LIN {X 0.195,Y -645.562,Z 909.524,A 0.000,B 0.000,C 90.000,E1 130.297} C_DIS
LIN {X -0.083,Y -651.299,Z 909.516,A 0.000,B 0.000,C 90.000,E1 128.830} C_DIS
LIN {X 0.215,Y -657.933,Z 909.506,A 0.000,B 0.000,C 90.000,E1 127.076} C_DIS
LIN {X -0.215,Y -660.619,Z 909.502,A 0.000,B 0.000,C 90.000,E1 126.377} C_DIS
LIN {X -0.067,Y -665.794,Z 909.494,A 0.000,B 0.000,C 90.000,E1 124.898} C_DIS
LIN {X 0.087,Y -669.096,Z 909.488,A 0.000,B 0.000,C 90.000,E1 123.913} C_DIS
LIN {X 0.321,Y -671.422,Z 909.484,A 0.000,B 0.000,C 90.000,E1 123.166} C_DIS
LIN {X 0.173,Y -674.186,Z 909.479,A 0.000,B 0.000,C 90.000,E1 122.212} C_DIS
LIN {X 0.234,Y -677.133,Z 909.472,A 0.000,B 0.000,C 90.000,E1 121.003} C_DIS
LIN {X -0.193,Y -679.151,Z 909.467,A 0.000,B 0.000,C 90.000,E1 120.079} C_DIS
LIN {X 0.332,Y -680.834,Z 909.462,A 0.000,B 0.000,C 90.000,E1 119.077} C_DIS
LIN {X 0.338,Y -682.009,Z 909.458,A 0.000,B 0.000,C 90.000,E1 118.359} C_DIS
LIN {X -0.041,Y -683.207,Z 909.452,A 0.000,B 0.000,C 90.000,E1 117.436} C_DIS
LIN {X -0.114,Y -683.928,Z 909.447,A 0.000,B 0.000,C 90.000,E1 116.488} C_DIS
LIN {X 0.047,Y -684.370,Z 909.441,A 0.000,B 0.000,C 90.000,E1 115.283} C_DIS
LIN {X -0.001,Y -684.293,Z 909.435,A 0.000,B 0.000,C 90.000,E1 114.335} C_DIS
LIN {X 0.425,Y -684.073,Z 909.433,A 0.000,B 0.000,C 90.000,E1 113.823} C_DIS
LIN {X -0.265,Y -683.873,Z 909.431,A 0.000,B 0.000,C 90.000,E1 113.643} C_DIS
LIN {X 0.153,Y -683.084,Z 909.429,A 0.000,B 0.000,C 90.000,E1 113.131} C_DIS
LIN {X 0.093,Y -682.298,Z 909.427,A 0.000,B 0.000,C 90.000,E1 112.898} C_DIS
LIN {X -0.391,Y -680.091,Z 909.425,A 0.000,B 0.000,C 90.000,E1 112.461} C_DIS
LIN {X -0.292,Y -679.235,Z 909.424,A 0.000,B 0.000,C 90.000,E1 112.333} C_DIS
LIN {X -0.194,Y -677.946,Z 909.423,A 0.000,B 0.000,C 90.000,E1 112.206} C_DIS
LIN {X -0.045,Y -676.193,Z 909.423,A 0.000,B 0.000,C 90.000,E1 112.078} C_DIS
LIN {X 0.034,Y -673.633,Z 909.421,A 0.000,B 0.000,C 90.000,E1 111.844} C_DIS
LIN {X 0.216,Y -672.143,Z 909.421,A 0.000,B 0.000,C 90.000,E1 111.716} C_DIS
LIN {X -0.131,Y -669.831,Z 909.420,A 0.000,B 0.000,C 90.000,E1 111.642} C_DIS
LIN {X 0.163,Y -662.934,Z 909.419,A 0.000,B 0.000,C 90.000,E1 111.408} C_DIS
LIN {X 0.168,Y -660.795,Z 909.419,A 0.000,B 0.000,C 90.000,E1 111.354} C_DIS
LIN {X -0.046,Y -652.097,Z 909.418,A 0.000,B 0.000,C 90.000,E1 111.280} C_DIS
LIN {X 0.172,Y -639.351,Z 909.418,A 0.000,B 0.000,C 90.000,E1 111.153} C_DIS
LIN {X -0.202,Y -633.090,Z 909.417,A 0.000,B 0.000,C 90.000,E1 111.099} C_DIS
LIN {X -0.001,Y -627.196,Z 909.417,A 0.000,B 0.000,C 90.000,E1 110.972} C_DIS
LIN {X -0.005,Y -619.742,Z 909.416,A 0.000,B 0.000,C 90.000,E1 110.791} C_DIS
LIN {X 0.025,Y -612.472,Z 909.414,A 0.000,B 0.000,C 90.000,E1 110.556} C_DIS
LIN {X 0.234,Y -605.407,Z 909.413,A 0.000,B 0.000,C 90.000,E1 110.248} C_DIS
LIN {X -0.232,Y -599.446,Z 909.411,A 0.000,B 0.000,C 90.000,E1 109.993} C_DIS
LIN {X 0.123,Y -581.326,Z 909.405,A 0.000,B 0.000,C 90.000,E1 108.852} C_DIS
LIN {X 0.041,Y -577.804,Z 909.404,A 0.000,B 0.000,C 90.000,E1 108.671} C_DIS
LIN {X 0.004,Y -572.696,Z 909.402,A 0.000,B 0.000,C 90.000,E1 108.417} C_DIS
LIN {X -0.230,Y -557.264,Z 909.399,A 0.000,B 0.000,C 90.000,E1 107.819} C_DIS
LIN {X -0.214,Y -556.236,Z 909.399,A 0.000,B 0.000,C 90.000,E1 107.764} C_DIS
LIN {X -0.009,Y -554.802,Z 909.398,A 0.000,B 0.000,C 90.000,E1 107.583} C_DIS
LIN {X -0.049,Y -554.765,Z 909.398,A 0.000,B 0.000,C 90.000,E1 107.583} C_DIS
LIN {X -0.204,Y -554.317,Z 909.396,A 0.000,B 0.000,C 90.000,E1 107.330} C_DIS
LIN {X -0.152,Y -555.407,Z 909.377,A 0.000,B 0.000,C 90.000,E1 103.939} C_DIS
LIN {X 0.224,Y -556.528,Z 909.367,A 0.000,B 0.000,C 90.000,E1 101.951} C_DIS
LIN {X 0.090,Y -557.923,Z 909.356,A 0.000,B 0.000,C 90.000,E1 100.018} C_DIS
LIN {X 0.201,Y -559.105,Z 909.346,A 0.000,B 0.000,C 90.000,E1 98.341} C_DIS
LIN {X 0.275,Y -560.081,Z 909.339,A 0.000,B 0.000,C 90.000,E1 96.947} C_DIS
LIN {X -0.112,Y -561.212,Z 909.328,A 0.000,B 0.000,C 90.000,E1 95.049} C_DIS
LIN {X -0.136,Y -561.882,Z 909.320,A 0.000,B 0.000,C 90.000,E1 93.669} C_DIS
LIN {X -0.082,Y -562.613,Z 909.311,A 0.000,B 0.000,C 90.000,E1 92.007} C_DIS
LIN {X -0.117,Y -563.071,Z 909.303,A 0.000,B 0.000,C 90.000,E1 90.630} C_DIS
LIN {X -0.158,Y -563.456,Z 909.296,A 0.000,B 0.000,C 90.000,E1 89.255} C_DIS
LIN {X -0.073,Y -563.806,Z 909.287,A 0.000,B 0.000,C 90.000,E1 87.593} C_DIS
LIN {X 0.151,Y -564.119,Z 909.276,A 0.000,B 0.000,C 90.000,E1 85.641} C_DIS
LIN {X -0.290,Y -564.432,Z 909.267,A 0.000,B 0.000,C 90.000,E1 84.033} C_DIS
LIN {X 0.199,Y -564.884,Z 909.255,A 0.000,B 0.000,C 90.000,E1 81.781} C_DIS
LIN {X 0.223,Y -565.616,Z 909.242,A 0.000,B 0.000,C 90.000,E1 79.577} C_DIS
LIN {X -0.247,Y -566.559,Z 909.232,A 0.000,B 0.000,C 90.000,E1 77.701} C_DIS
LIN {X -0.007,Y -567.553,Z 909.221,A 0.000,B 0.000,C 90.000,E1 75.755} C_DIS
LIN {X 0.283,Y -568.145,Z 909.215,A 0.000,B 0.000,C 90.000,E1 74.629} C_DIS
LIN {X -0.013,Y -568.893,Z 909.206,A 0.000,B 0.000,C 90.000,E1 73.015} C_DIS
LIN {X 0.078,Y -569.455,Z 909.198,A 0.000,B 0.000,C 90.000,E1 71.638} C_DIS
LIN {X -0.184,Y -569.869,Z 909.190,A 0.000,B 0.000,C 90.000,E1 70.296} C_DIS
LIN {X 0.098,Y -570.165,Z 909.183,A 0.000,B 0.000,C 90.000,E1 68.901} C_DIS
LIN {X 0.230,Y -570.417,Z 909.177,A 0.000,B 0.000,C 90.000,E1 67.794} C_DIS
LIN {X 0.011,Y -570.638,Z 909.168,A 0.000,B 0.000,C 90.000,E1 66.177} C_DIS
LIN {X 0.027,Y -570.717,Z 909.159,A 0.000,B 0.000,C 90.000,E1 64.537} C_DIS
LIN {X -0.048,Y -570.753,Z 909.151,A 0.000,B 0.000,C 90.000,E1 63.179} C_DIS
LIN {X -0.114,Y -570.728,Z 909.143,A 0.000,B 0.000,C 90.000,E1 61.820} C_DIS
LIN {X 0.247,Y -570.545,Z 909.133,A 0.000,B 0.000,C 90.000,E1 59.871} C_DIS
LIN {X 0.070,Y -570.097,Z 909.124,A 0.000,B 0.000,C 90.000,E1 58.250} C_DIS
LIN {X -0.172,Y -569.741,Z 909.119,A 0.000,B 0.000,C 90.000,E1 57.454} C_DIS
LIN {X -0.182,Y -569.052,Z 909.112,A 0.000,B 0.000,C 90.000,E1 56.087} C_DIS
LIN {X 0.114,Y -568.040,Z 909.104,A 0.000,B 0.000,C 90.000,E1 54.689} C_DIS
LIN {X -0.189,Y -567.032,Z 909.098,A 0.000,B 0.000,C 90.000,E1 53.623} C_DIS
LIN {X -0.046,Y -565.386,Z 909.090,A 0.000,B 0.000,C 90.000,E1 52.236} C_DIS
LIN {X -0.057,Y -564.293,Z 909.086,A 0.000,B 0.000,C 90.000,E1 51.412} C_DIS
LIN {X -0.177,Y -563.017,Z 909.081,A 0.000,B 0.000,C 90.000,E1 50.598} C_DIS
LIN {X 0.147,Y -560.951,Z 909.075,A 0.000,B 0.000,C 90.000,E1 49.461} C_DIS
LIN {X -0.095,Y -559.868,Z 909.072,A 0.000,B 0.000,C 90.000,E1 48.933} C_DIS
LIN {X 0.106,Y -557.972,Z 909.067,A 0.000,B 0.000,C 90.000,E1 48.081} C_DIS
LIN {X 0.287,Y -555.739,Z 909.063,A 0.000,B 0.000,C 90.000,E1 47.229} C_DIS
LIN {X 0.006,Y -554.137,Z 909.060,A 0.000,B 0.000,C 90.000,E1 46.701} C_DIS
LIN {X -0.257,Y -551.428,Z 909.055,A 0.000,B 0.000,C 90.000,E1 45.891} C_DIS
LIN {X 0.232,Y -548.426,Z 909.050,A 0.000,B 0.000,C 90.000,E1 45.000} C_DIS
LIN {X -0.086,Y -545.106,Z 909.045,A 0.000,B 0.000,C 90.000,E1 44.190} C_DIS
LIN {X -0.258,Y -543.280,Z 909.043,A 0.000,B 0.000,C 90.000,E1 43.785} C_DIS
LIN {X -0.242,Y -539.229,Z 909.038,A 0.000,B 0.000,C 90.000,E1 42.933} C_DIS
LIN {X 0.313,Y -537.097,Z 909.036,A 0.000,B 0.000,C 90.000,E1 42.447} C_DIS
LIN {X -0.090,Y -534.054,Z 909.033,A 0.000,B 0.000,C 90.000,E1 41.919} C_DIS
LIN {X 0.008,Y -529.937,Z 909.029,A 0.000,B 0.000,C 90.000,E1 41.191} C_DIS
LIN {X -0.040,Y -526.414,Z 909.026,A 0.000,B 0.000,C 90.000,E1 40.620} C_DIS
LIN {X 0.042,Y -521.743,Z 909.022,A 0.000,B 0.000,C 90.000,E1 39.886} C_DIS
LIN {X -0.185,Y -515.782,Z 909.017,A 0.000,B 0.000,C 90.000,E1 39.036} C_DIS
LIN {X -0.320,Y -511.502,Z 909.014,A 0.000,B 0.000,C 90.000,E1 38.463} C_DIS
LIN {X 0.137,Y -508.167,Z 909.011,A 0.000,B 0.000,C 90.000,E1 37.971} C_DIS
LIN {X -0.029,Y -503.410,Z 909.008,A 0.000,B 0.000,C 90.000,E1 37.397} C_DIS
LIN {X -0.153,Y -497.100,Z 909.004,A 0.000,B 0.000,C 90.000,E1 36.664} C_DIS
LIN {X 0.175,Y -490.367,Z 909.000,A 0.000,B 0.000,C 90.000,E1 35.884} C_DIS
LIN {X 0.211,Y -484.732,Z 908.996,A 0.000,B 0.000,C 90.000,E1 35.311} C_DIS
LIN {X 0.108,Y -479.044,Z 908.993,A 0.000,B 0.000,C 90.000,E1 34.771} C_DIS
LIN {X -0.082,Y -473.038,Z 908.990,A 0.000,B 0.000,C 90.000,E1 34.246} C_DIS
LIN {X -0.054,Y -464.073,Z 908.986,A 0.000,B 0.000,C 90.000,E1 33.452} C_DIS
LIN {X -0.014,Y -453.438,Z 908.981,A 0.000,B 0.000,C 90.000,E1 32.546} C_DIS
LIN {X -0.187,Y -442.578,Z 908.976,A 0.000,B 0.000,C 90.000,E1 31.671} C_DIS
LIN {X 0.065,Y -431.669,Z 908.971,A 0.000,B 0.000,C 90.000,E1 30.747} C_DIS
LIN {X -0.085,Y -409.120,Z 908.960,A 0.000,B 0.000,C 90.000,E1 28.743} C_DIS
LIN {X -0.133,Y -398.923,Z 908.954,A 0.000,B 0.000,C 90.000,E1 27.719} C_DIS
LIN {X 0.086,Y -394.402,Z 908.951,A 0.000,B 0.000,C 90.000,E1 27.129} C_DIS
LIN {X -0.030,Y -393.388,Z 908.950,A 0.000,B 0.000,C 90.000,E1 27.001} C_DIS
LIN {X 0.106,Y -390.640,Z 908.947,A 0.000,B 0.000,C 90.000,E1 26.437} C_DIS
LIN {X -0.083,Y -389.421,Z 908.944,A 0.000,B 0.000,C 90.000,E1 25.976} C_DIS
LIN {X -0.231,Y -388.825,Z 908.940,A 0.000,B 0.000,C 90.000,E1 25.283} C_DIS
LIN {X 0.138,Y -388.845,Z 908.936,A 0.000,B 0.000,C 90.000,E1 24.515} C_DIS
LIN {X 0.201,Y -389.687,Z 908.928,A 0.000,B 0.000,C 90.000,E1 23.078} C_DIS
LIN {X -0.187,Y -393.165,Z 908.909,A 0.000,B 0.000,C 90.000,E1 19.577} C_DIS
LIN {X -0.094,Y -396.472,Z 908.893,A 0.000,B 0.000,C 90.000,E1 16.732} C_DIS
LIN {X 0.070,Y -399.567,Z 908.879,A 0.000,B 0.000,C 90.000,E1 14.245} C_DIS
LIN {X -0.159,Y -403.025,Z 908.866,A 0.000,B 0.000,C 90.000,E1 11.827} C_DIS
LIN {X -0.061,Y -407.346,Z 908.850,A 0.000,B 0.000,C 90.000,E1 9.029} C_DIS
LIN {X -0.030,Y -411.518,Z 908.837,A 0.000,B 0.000,C 90.000,E1 6.606} C_DIS
LIN {X 0.125,Y -416.684,Z 908.821,A 0.000,B 0.000,C 90.000,E1 3.841} C_DIS
LIN {X -0.058,Y -422.526,Z 908.806,A 0.000,B 0.000,C 90.000,E1 1.146} C_DIS
LIN {X 0.190,Y -431.613,Z 908.786,A 0.000,B 0.000,C 90.000,E1 357.421} C_DIS
LIN {X -0.066,Y -433.865,Z 908.782,A 0.000,B 0.000,C 90.000,E1 356.788} C_DIS
LIN {X 0.060,Y -436.175,Z 908.779,A 0.000,B 0.000,C 90.000,E1 356.274} C_DIS
LIN {X 0.105,Y -437.112,Z 908.778,A 0.000,B 0.000,C 90.000,E1 356.102} C_DIS
LIN {X 0.134,Y -440.525,Z 908.776,A 0.000,B 0.000,C 90.000,E1 355.698} C_DIS
LIN {X -0.211,Y -442.095,Z 908.775,A 0.000,B 0.000,C 90.000,E1 355.584} C_DIS
LIN {X 0.084,Y -447.635,Z 908.773,A 0.000,B 0.000,C 90.000,E1 355.179} C_DIS
LIN {X -0.204,Y -462.189,Z 908.770,A 0.000,B 0.000,C 90.000,E1 354.546} C_DIS
LIN {X 0.073,Y -475.661,Z 908.766,A 0.000,B 0.000,C 90.000,E1 353.856} C_DIS
LIN {X 0.119,Y -485.730,Z 908.763,A 0.000,B 0.000,C 90.000,E1 353.337} C_DIS
LIN {X 0.093,Y -500.234,Z 908.759,A 0.000,B 0.000,C 90.000,E1 352.534} C_DIS
LIN {X 0.201,Y -508.278,Z 908.756,A 0.000,B 0.000,C 90.000,E1 352.064} C_DIS
LIN {X 0.031,Y -517.662,Z 908.753,A 0.000,B 0.000,C 90.000,E1 351.489} C_DIS
LIN {X 0.171,Y -526.953,Z 908.749,A 0.000,B 0.000,C 90.000,E1 350.849} C_DIS
LIN {X -0.134,Y -532.964,Z 908.747,A 0.000,B 0.000,C 90.000,E1 350.443} C_DIS
LIN {X -0.124,Y -538.715,Z 908.744,A 0.000,B 0.000,C 90.000,E1 349.982} C_DIS
LIN {X 0.185,Y -545.677,Z 908.741,A 0.000,B 0.000,C 90.000,E1 349.342} C_DIS
LIN {X 0.165,Y -552.370,Z 908.737,A 0.000,B 0.000,C 90.000,E1 348.701} C_DIS
LIN {X 0.033,Y -558.750,Z 908.734,A 0.000,B 0.000,C 90.000,E1 348.049} C_DIS
LIN {X -0.138,Y -563.608,Z 908.731,A 0.000,B 0.000,C 90.000,E1 347.521} C_DIS
LIN {X -0.184,Y -570.490,Z 908.726,A 0.000,B 0.000,C 90.000,E1 346.700} C_DIS
LIN {X 0.077,Y -575.709,Z 908.722,A 0.000,B 0.000,C 90.000,E1 345.992} C_DIS
LIN {X -0.070,Y -579.705,Z 908.719,A 0.000,B 0.000,C 90.000,E1 345.463} C_DIS
LIN {X -0.144,Y -586.930,Z 908.713,A 0.000,B 0.000,C 90.000,E1 344.393} C_DIS
LIN {X -0.301,Y -591.105,Z 908.710,A 0.000,B 0.000,C 90.000,E1 343.740} C_DIS
LIN {X -0.047,Y -597.242,Z 908.704,A 0.000,B 0.000,C 90.000,E1 342.653} C_DIS
LIN {X 0.113,Y -602.926,Z 908.698,A 0.000,B 0.000,C 90.000,E1 341.583} C_DIS
LIN {X -0.074,Y -608.917,Z 908.691,A 0.000,B 0.000,C 90.000,E1 340.423} C_DIS
LIN {X -0.120,Y -613.345,Z 908.686,A 0.000,B 0.000,C 90.000,E1 339.518} C_DIS
LIN {X 0.097,Y -617.537,Z 908.681,A 0.000,B 0.000,C 90.000,E1 338.592} C_DIS
LIN {X 0.110,Y -623.248,Z 908.674,A 0.000,B 0.000,C 90.000,E1 337.305} C_DIS
LIN {X -0.133,Y -627.339,Z 908.668,A 0.000,B 0.000,C 90.000,E1 336.305} C_DIS
LIN {X -0.060,Y -631.107,Z 908.663,A 0.000,B 0.000,C 90.000,E1 335.281} C_DIS
LIN {X -0.198,Y -634.766,Z 908.657,A 0.000,B 0.000,C 90.000,E1 334.280} C_DIS
LIN {X -0.066,Y -637.407,Z 908.653,A 0.000,B 0.000,C 90.000,E1 333.512} C_DIS
LIN {X 0.094,Y -639.777,Z 908.649,A 0.000,B 0.000,C 90.000,E1 332.743} C_DIS
LIN {X -0.225,Y -642.799,Z 908.643,A 0.000,B 0.000,C 90.000,E1 331.769} C_DIS
LIN {X 0.371,Y -645.562,Z 908.638,A 0.000,B 0.000,C 90.000,E1 330.717} C_DIS
LIN {X -0.357,Y -648.851,Z 908.631,A 0.000,B 0.000,C 90.000,E1 329.537} C_DIS
LIN {X -0.155,Y -651.906,Z 908.624,A 0.000,B 0.000,C 90.000,E1 328.280} C_DIS
LIN {X -0.096,Y -653.633,Z 908.620,A 0.000,B 0.000,C 90.000,E1 327.533} C_DIS
LIN {X -0.023,Y -655.966,Z 908.613,A 0.000,B 0.000,C 90.000,E1 326.294} C_DIS
LIN {X 0.074,Y -657.235,Z 908.609,A 0.000,B 0.000,C 90.000,E1 325.548} C_DIS
LIN {X 0.043,Y -658.966,Z 908.602,A 0.000,B 0.000,C 90.000,E1 324.322} C_DIS
LIN {X -0.338,Y -660.459,Z 908.595,A 0.000,B 0.000,C 90.000,E1 323.130} C_DIS
LIN {X 0.178,Y -661.956,Z 908.587,A 0.000,B 0.000,C 90.000,E1 321.618} C_DIS
LIN {X 0.177,Y -663.531,Z 908.577,A 0.000,B 0.000,C 90.000,E1 319.908} C_DIS
LIN {X 0.182,Y -665.606,Z 908.565,A 0.000,B 0.000,C 90.000,E1 317.715} C_DIS
LIN {X -0.293,Y -666.828,Z 908.558,A 0.000,B 0.000,C 90.000,E1 316.539} C_DIS
LIN {X -0.290,Y -667.514,Z 908.554,A 0.000,B 0.000,C 90.000,E1 315.810} C_DIS
LIN {X -0.253,Y -669.043,Z 908.545,A 0.000,B 0.000,C 90.000,E1 314.109} C_DIS
LIN {X 0.296,Y -670.591,Z 908.536,A 0.000,B 0.000,C 90.000,E1 312.366} C_DIS
LIN {X 0.400,Y -671.731,Z 908.529,A 0.000,B 0.000,C 90.000,E1 311.148} C_DIS
LIN {X 0.098,Y -672.889,Z 908.521,A 0.000,B 0.000,C 90.000,E1 309.725} C_DIS
LIN {X -0.191,Y -673.865,Z 908.514,A 0.000,B 0.000,C 90.000,E1 308.543} C_DIS
LIN {X 0.064,Y -674.800,Z 908.507,A 0.000,B 0.000,C 90.000,E1 307.317} C_DIS
LIN {X -0.207,Y -675.377,Z 908.502,A 0.000,B 0.000,C 90.000,E1 306.377} C_DIS
LIN {X 0.214,Y -676.122,Z 908.494,A 0.000,B 0.000,C 90.000,E1 304.898} C_DIS
LIN {X -0.296,Y -676.820,Z 908.486,A 0.000,B 0.000,C 90.000,E1 303.499} C_DIS
LIN {X -0.064,Y -677.837,Z 908.477,A 0.000,B 0.000,C 90.000,E1 301.799} C_DIS
LIN {X 0.028,Y -679.350,Z 908.466,A 0.000,B 0.000,C 90.000,E1 299.873} C_DIS
LIN {X 0.257,Y -682.866,Z 908.449,A 0.000,B 0.000,C 90.000,E1 296.744} C_DIS
LIN {X 0.145,Y -685.537,Z 908.438,A 0.000,B 0.000,C 90.000,E1 294.847} C_DIS
LIN {X 0.116,Y -686.627,Z 908.433,A 0.000,B 0.000,C 90.000,E1 293.898} C_DIS
LIN {X -0.075,Y -687.047,Z 908.430,A 0.000,B 0.000,C 90.000,E1 293.439} C_DIS
LIN {X 0.093,Y -687.264,Z 908.428,A 0.000,B 0.000,C 90.000,E1 292.950} C_DIS
LIN {X 0.265,Y -686.844,Z 908.425,A 0.000,B 0.000,C 90.000,E1 292.461} C_DIS
LIN {X -0.153,Y -686.411,Z 908.424,A 0.000,B 0.000,C 90.000,E1 292.259} C_DIS
LIN {X 0.015,Y -684.112,Z 908.421,A 0.000,B 0.000,C 90.000,E1 291.770} C_DIS
LIN {X -0.029,Y -682.572,Z 908.420,A 0.000,B 0.000,C 90.000,E1 291.535} C_DIS
LIN {X 0.071,Y -681.425,Z 908.419,A 0.000,B 0.000,C 90.000,E1 291.408} C_DIS
LIN {X 0.170,Y -679.661,Z 908.418,A 0.000,B 0.000,C 90.000,E1 291.280} C_DIS
LIN {X 0.158,Y -672.887,Z 908.416,A 0.000,B 0.000,C 90.000,E1 290.918} C_DIS
LIN {X 0.153,Y -665.738,Z 908.415,A 0.000,B 0.000,C 90.000,E1 290.610} C_DIS
LIN {X 0.151,Y -661.194,Z 908.413,A 0.000,B 0.000,C 90.000,E1 290.375} C_DIS
LIN {X 0.091,Y -661.149,Z 908.413,A 0.000,B 0.000,C 90.000,E1 290.375} C_DIS
LIN {X -0.048,Y -660.567,Z 908.413,A 0.000,B 0.000,C 90.000,E1 290.301} C_DIS
LIN {X -0.093,Y -660.547,Z 908.413,A 0.000,B 0.000,C 90.000,E1 290.301} C_DIS
LIN {X 0.061,Y -660.564,Z 908.412,A 0.000,B 0.000,C 90.000,E1 290.066} C_DIS
LIN {X 0.064,Y -662.013,Z 908.409,A 0.000,B 0.000,C 90.000,E1 289.577} C_DIS
LIN {X 0.151,Y -664.034,Z 908.406,A 0.000,B 0.000,C 90.000,E1 289.087} C_DIS
LIN {X 0.047,Y -671.509,Z 908.398,A 0.000,B 0.000,C 90.000,E1 287.638} C_DIS
LIN {X -0.090,Y -673.798,Z 908.395,A 0.000,B 0.000,C 90.000,E1 287.166} C_DIS
LIN {X -0.072,Y -676.837,Z 908.391,A 0.000,B 0.000,C 90.000,E1 286.441} C_DIS
LIN {X -0.031,Y -679.173,Z 908.387,A 0.000,B 0.000,C 90.000,E1 285.717} C_DIS
LIN {X -0.117,Y -680.451,Z 908.385,A 0.000,B 0.000,C 90.000,E1 285.245} C_DIS
LIN {X -0.287,Y -683.062,Z 908.378,A 0.000,B 0.000,C 90.000,E1 284.064} C_DIS
LIN {X 0.297,Y -684.275,Z 908.374,A 0.000,B 0.000,C 90.000,E1 283.300} C_DIS
LIN {X 0.205,Y -685.582,Z 908.369,A 0.000,B 0.000,C 90.000,E1 282.355} C_DIS
LIN {X 0.000,Y -686.195,Z 908.365,A 0.000,B 0.000,C 90.000,E1 281.658} C_DIS
LIN {X -0.039,Y -686.413,Z 908.362,A 0.000,B 0.000,C 90.000,E1 281.186} C_DIS
LIN {X -0.082,Y -686.381,Z 908.360,A 0.000,B 0.000,C 90.000,E1 280.715} C_DIS
LIN {X -0.251,Y -685.980,Z 908.357,A 0.000,B 0.000,C 90.000,E1 280.254} C_DIS
LIN {X -0.275,Y -685.653,Z 908.356,A 0.000,B 0.000,C 90.000,E1 280.018} C_DIS
LIN {X 0.232,Y -684.729,Z 908.353,A 0.000,B 0.000,C 90.000,E1 279.500} C_DIS
LIN {X 0.170,Y -683.507,Z 908.350,A 0.000,B 0.000,C 90.000,E1 279.029} C_DIS
LIN {X -0.008,Y -681.823,Z 908.348,A 0.000,B 0.000,C 90.000,E1 278.568} C_DIS
LIN {X -0.194,Y -679.778,Z 908.345,A 0.000,B 0.000,C 90.000,E1 278.106} C_DIS
LIN {X 0.223,Y -676.392,Z 908.341,A 0.000,B 0.000,C 90.000,E1 277.352} C_DIS
LIN {X -0.075,Y -673.192,Z 908.338,A 0.000,B 0.000,C 90.000,E1 276.777} C_DIS
LIN {X 0.271,Y -669.663,Z 908.334,A 0.000,B 0.000,C 90.000,E1 276.144} C_DIS
LIN {X 0.093,Y -667.413,Z 908.332,A 0.000,B 0.000,C 90.000,E1 275.796} C_DIS
LIN {X -0.272,Y -663.096,Z 908.329,A 0.000,B 0.000,C 90.000,E1 275.220} C_DIS
LIN {X 0.081,Y -659.326,Z 908.326,A 0.000,B 0.000,C 90.000,E1 274.702} C_DIS
LIN {X -0.299,Y -655.183,Z 908.323,A 0.000,B 0.000,C 90.000,E1 274.245} C_DIS
LIN {X -0.107,Y -649.293,Z 908.320,A 0.000,B 0.000,C 90.000,E1 273.612} C_DIS
LIN {X 0.291,Y -644.297,Z 908.317,A 0.000,B 0.000,C 90.000,E1 273.094} C_DIS
LIN {X 0.278,Y -637.563,Z 908.314,A 0.000,B 0.000,C 90.000,E1 272.522} C_DIS
LIN {X -0.070,Y -630.336,Z 908.311,A 0.000,B 0.000,C 90.000,E1 272.007} C_DIS
LIN {X -0.095,Y -624.332,Z 908.309,A 0.000,B 0.000,C 90.000,E1 271.604} C_DIS
LIN {X 0.089,Y -618.139,Z 908.307,A 0.000,B 0.000,C 90.000,E1 271.203} C_DIS
LIN {X 0.255,Y -609.882,Z 908.304,A 0.000,B 0.000,C 90.000,E1 270.745} C_DIS
LIN {X -0.185,Y -603.169,Z 908.302,A 0.000,B 0.000,C 90.000,E1 270.458} C_DIS
LIN {X -0.219,Y -598.145,Z 908.301,A 0.000,B 0.000,C 90.000,E1 270.229} C_DIS
LIN {X -0.149,Y -590.978,Z 908.300,A 0.000,B 0.000,C 90.000,E1 269.943} C_DIS
LIN {X 0.259,Y -583.781,Z 908.298,A 0.000,B 0.000,C 90.000,E1 269.656} C_DIS
LIN {X -0.249,Y -578.196,Z 908.297,A 0.000,B 0.000,C 90.000,E1 269.542} C_DIS
LIN {X 0.036,Y -571.792,Z 908.297,A 0.000,B 0.000,C 90.000,E1 269.370} C_DIS
LIN {X 0.144,Y -565.261,Z 908.296,A 0.000,B 0.000,C 90.000,E1 269.255} C_DIS
LIN {X -0.224,Y -554.852,Z 908.295,A 0.000,B 0.000,C 90.000,E1 269.198} C_DIS
LIN {X 0.157,Y -552.543,Z 908.295,A 0.000,B 0.000,C 90.000,E1 269.141} C_DIS
LIN {X -0.136,Y -549.494,Z 908.295,A 0.000,B 0.000,C 90.000,E1 269.083} C_DIS
LIN {X -0.168,Y -549.414,Z 908.295,A 0.000,B 0.000,C 90.000,E1 269.083} C_DIS
LIN {X 0.187,Y -545.395,Z 908.293,A 0.000,B 0.000,C 90.000,E1 268.682} C_DIS
LIN {X 0.150,Y -545.361,Z 908.293,A 0.000,B 0.000,C 90.000,E1 268.682} C_DIS
LIN {X 0.055,Y -544.265,Z 908.291,A 0.000,B 0.000,C 90.000,E1 268.396} C_DIS
LIN {X -0.029,Y -543.383,Z 908.288,A 0.000,B 0.000,C 90.000,E1 267.822} C_DIS
LIN {X -0.155,Y -540.427,Z 908.269,A 0.000,B 0.000,C 90.000,E1 264.432} C_DIS
LIN {X -0.017,Y -539.422,Z 908.261,A 0.000,B 0.000,C 90.000,E1 262.996} C_DIS
LIN {X 0.167,Y -538.477,Z 908.255,A 0.000,B 0.000,C 90.000,E1 261.837} C_DIS
LIN {X -0.128,Y -537.130,Z 908.247,A 0.000,B 0.000,C 90.000,E1 260.443} C_DIS
LIN {X 0.020,Y -535.946,Z 908.241,A 0.000,B 0.000,C 90.000,E1 259.285} C_DIS
LIN {X 0.190,Y -535.031,Z 908.236,A 0.000,B 0.000,C 90.000,E1 258.409} C_DIS
LIN {X 0.046,Y -533.384,Z 908.228,A 0.000,B 0.000,C 90.000,E1 256.992} C_DIS
LIN {X -0.077,Y -531.258,Z 908.218,A 0.000,B 0.000,C 90.000,E1 255.283} C_DIS
LIN {X 0.079,Y -528.397,Z 908.205,A 0.000,B 0.000,C 90.000,E1 252.960} C_DIS
LIN {X 0.120,Y -526.617,Z 908.197,A 0.000,B 0.000,C 90.000,E1 251.511} C_DIS
LIN {X 0.294,Y -524.330,Z 908.188,A 0.000,B 0.000,C 90.000,E1 249.752} C_DIS
LIN {X 0.273,Y -522.809,Z 908.181,A 0.000,B 0.000,C 90.000,E1 248.592} C_DIS
LIN {X -0.107,Y -520.766,Z 908.173,A 0.000,B 0.000,C 90.000,E1 247.177} C_DIS
LIN {X 0.006,Y -519.133,Z 908.167,A 0.000,B 0.000,C 90.000,E1 245.997} C_DIS
LIN {X 0.117,Y -515.655,Z 908.154,A 0.000,B 0.000,C 90.000,E1 243.640} C_DIS
LIN {X -0.093,Y -512.723,Z 908.144,A 0.000,B 0.000,C 90.000,E1 241.897} C_DIS
LIN {X -0.104,Y -510.600,Z 908.137,A 0.000,B 0.000,C 90.000,E1 240.717} C_DIS
LIN {X 0.138,Y -506.936,Z 908.126,A 0.000,B 0.000,C 90.000,E1 238.614} C_DIS
LIN {X -0.138,Y -504.719,Z 908.119,A 0.000,B 0.000,C 90.000,E1 237.454} C_DIS
LIN {X 0.254,Y -502.306,Z 908.112,A 0.000,B 0.000,C 90.000,E1 236.215} C_DIS
LIN {X 0.032,Y -500.378,Z 908.108,A 0.000,B 0.000,C 90.000,E1 235.341} C_DIS
LIN {X 0.230,Y -497.545,Z 908.101,A 0.000,B 0.000,C 90.000,E1 234.116} C_DIS
LIN {X 0.099,Y -494.880,Z 908.094,A 0.000,B 0.000,C 90.000,E1 232.924} C_DIS
LIN {X 0.069,Y -491.502,Z 908.086,A 0.000,B 0.000,C 90.000,E1 231.412} C_DIS
LIN {X -0.114,Y -486.769,Z 908.074,A 0.000,B 0.000,C 90.000,E1 229.299} C_DIS
LIN {X 0.002,Y -484.753,Z 908.069,A 0.000,B 0.000,C 90.000,E1 228.366} C_DIS
LIN {X 0.091,Y -479.245,Z 908.055,A 0.000,B 0.000,C 90.000,E1 225.891} C_DIS
LIN {X 0.003,Y -475.753,Z 908.046,A 0.000,B 0.000,C 90.000,E1 224.352} C_DIS
LIN {X 0.188,Y -472.164,Z 908.038,A 0.000,B 0.000,C 90.000,E1 222.771} C_DIS
LIN {X -0.176,Y -467.264,Z 908.026,A 0.000,B 0.000,C 90.000,E1 220.620} C_DIS
LIN {X -0.122,Y -463.916,Z 908.017,A 0.000,B 0.000,C 90.000,E1 219.036} C_DIS
LIN {X 0.046,Y -459.878,Z 908.006,A 0.000,B 0.000,C 90.000,E1 217.111} C_DIS
LIN {X 0.025,Y -456.526,Z 907.997,A 0.000,B 0.000,C 90.000,E1 215.518} C_DIS
LIN {X 0.037,Y -453.105,Z 907.988,A 0.000,B 0.000,C 90.000,E1 213.913} C_DIS
LIN {X -0.030,Y -447.336,Z 907.974,A 0.000,B 0.000,C 90.000,E1 211.337} C_DIS
LIN {X 0.185,Y -445.182,Z 907.969,A 0.000,B 0.000,C 90.000,E1 210.335} C_DIS
LIN {X -0.076,Y -440.957,Z 907.958,A 0.000,B 0.000,C 90.000,E1 208.409} C_DIS
LIN {X 0.095,Y -437.328,Z 907.949,A 0.000,B 0.000,C 90.000,E1 206.744} C_DIS
LIN {X 0.018,Y -432.988,Z 907.938,A 0.000,B 0.000,C 90.000,E1 204.771} C_DIS
LIN {X 0.051,Y -428.640,Z 907.927,A 0.000,B 0.000,C 90.000,E1 202.770} C_DIS
LIN {X 0.021,Y -425.079,Z 907.917,A 0.000,B 0.000,C 90.000,E1 201.099} C_DIS
LIN {X -0.054,Y -420.844,Z 907.906,A 0.000,B 0.000,C 90.000,E1 199.087} C_DIS
LIN {X -0.127,Y -417.501,Z 907.897,A 0.000,B 0.000,C 90.000,E1 197.402} C_DIS
LIN {X -0.238,Y -413.381,Z 907.885,A 0.000,B 0.000,C 90.000,E1 195.371} C_DIS
LIN {X -0.044,Y -408.578,Z 907.872,A 0.000,B 0.000,C 90.000,E1 192.939} C_DIS
LIN {X 0.107,Y -405.900,Z 907.864,A 0.000,B 0.000,C 90.000,E1 191.535} C_DIS
LIN {X 0.144,Y -402.449,Z 907.855,A 0.000,B 0.000,C 90.000,E1 189.792} C_DIS
LIN {X 0.098,Y -398.212,Z 907.843,A 0.000,B 0.000,C 90.000,E1 187.701} C_DIS
LIN {X 0.070,Y -392.221,Z 907.825,A 0.000,B 0.000,C 90.000,E1 184.531} C_DIS
LIN {X -0.089,Y -388.034,Z 907.811,A 0.000,B 0.000,C 90.000,E1 182.064} C_DIS
LIN {X -0.170,Y -385.133,Z 907.802,A 0.000,B 0.000,C 90.000,E1 180.286} C_DIS
LIN {X -0.153,Y -381.252,Z 907.787,A 0.000,B 0.000,C 90.000,E1 177.764} C_DIS
LIN {X 0.031,Y -378.681,Z 907.777,A 0.000,B 0.000,C 90.000,E1 175.927} C_DIS
LIN {X 0.032,Y -377.484,Z 907.771,A 0.000,B 0.000,C 90.000,E1 174.837} C_DIS
LIN {X -0.056,Y -376.839,Z 907.763,A 0.000,B 0.000,C 90.000,E1 173.394} C_DIS
LIN {X 0.166,Y -376.923,Z 907.761,A 0.000,B 0.000,C 90.000,E1 172.996} C_DIS
LIN {X 0.060,Y -377.171,Z 907.759,A 0.000,B 0.000,C 90.000,E1 172.648} C_DIS
LIN {X -0.151,Y -378.296,Z 907.755,A 0.000,B 0.000,C 90.000,E1 171.951} C_DIS
LIN {X 0.123,Y -379.387,Z 907.753,A 0.000,B 0.000,C 90.000,E1 171.546} C_DIS
LIN {X -0.069,Y -381.425,Z 907.749,A 0.000,B 0.000,C 90.000,E1 170.849} C_DIS
LIN {X -0.180,Y -384.461,Z 907.746,A 0.000,B 0.000,C 90.000,E1 170.330} C_DIS
LIN {X 0.105,Y -387.519,Z 907.744,A 0.000,B 0.000,C 90.000,E1 169.859} C_DIS
LIN {X -0.121,Y -393.894,Z 907.740,A 0.000,B 0.000,C 90.000,E1 169.275} C_DIS
LIN {X 0.004,Y -401.829,Z 907.737,A 0.000,B 0.000,C 90.000,E1 168.701} C_DIS
LIN {X 0.222,Y -407.065,Z 907.735,A 0.000,B 0.000,C 90.000,E1 168.342} C_DIS
LIN {X -0.223,Y -418.459,Z 907.731,A 0.000,B 0.000,C 90.000,E1 167.645} C_DIS
LIN {X -0.041,Y -424.881,Z 907.729,A 0.000,B 0.000,C 90.000,E1 167.173} C_DIS
LIN {X 0.009,Y -431.295,Z 907.726,A 0.000,B 0.000,C 90.000,E1 166.700} C_DIS
LIN {X -0.224,Y -439.099,Z 907.723,A 0.000,B 0.000,C 90.000,E1 166.117} C_DIS
LIN {X -0.202,Y -452.668,Z 907.716,A 0.000,B 0.000,C 90.000,E1 164.936} C_DIS
LIN {X -0.153,Y -461.243,Z 907.712,A 0.000,B 0.000,C 90.000,E1 164.102} C_DIS
LIN {X -0.148,Y -470.949,Z 907.706,A 0.000,B 0.000,C 90.000,E1 163.087} C_DIS
LIN {X 0.175,Y -477.714,Z 907.702,A 0.000,B 0.000,C 90.000,E1 162.308} C_DIS
LIN {X 0.125,Y -482.805,Z 907.699,A 0.000,B 0.000,C 90.000,E1 161.710} C_DIS
LIN {X 0.173,Y -487.725,Z 907.695,A 0.000,B 0.000,C 90.000,E1 161.094} C_DIS
LIN {X 0.265,Y -490.296,Z 907.693,A 0.000,B 0.000,C 90.000,E1 160.786} C_DIS
LIN {X -0.013,Y -496.027,Z 907.689,A 0.000,B 0.000,C 90.000,E1 160.061} C_DIS
LIN {X 0.058,Y -504.825,Z 907.683,A 0.000,B 0.000,C 90.000,E1 158.847} C_DIS
LIN {X -0.238,Y -509.064,Z 907.679,A 0.000,B 0.000,C 90.000,E1 158.284} C_DIS
LIN {X -0.090,Y -514.004,Z 907.675,A 0.000,B 0.000,C 90.000,E1 157.539} C_DIS
LIN {X 0.107,Y -518.887,Z 907.671,A 0.000,B 0.000,C 90.000,E1 156.794} C_DIS
LIN {X 0.070,Y -524.800,Z 907.666,A 0.000,B 0.000,C 90.000,E1 155.921} C_DIS
LIN {X 0.209,Y -534.179,Z 907.658,A 0.000,B 0.000,C 90.000,E1 154.460} C_DIS
LIN {X 0.058,Y -541.158,Z 907.652,A 0.000,B 0.000,C 90.000,E1 153.332} C_DIS
LIN {X 0.263,Y -544.512,Z 907.649,A 0.000,B 0.000,C 90.000,E1 152.743} C_DIS
LIN {X -0.109,Y -548.599,Z 907.645,A 0.000,B 0.000,C 90.000,E1 152.076} C_DIS
LIN {X 0.184,Y -554.697,Z 907.639,A 0.000,B 0.000,C 90.000,E1 150.923} C_DIS
LIN {X -0.203,Y -559.100,Z 907.634,A 0.000,B 0.000,C 90.000,E1 150.127} C_DIS
LIN {X -0.077,Y -567.423,Z 907.625,A 0.000,B 0.000,C 90.000,E1 148.456} C_DIS
LIN {X -0.341,Y -571.372,Z 907.620,A 0.000,B 0.000,C 90.000,E1 147.661} C_DIS
LIN {X -0.349,Y -575.922,Z 907.615,A 0.000,B 0.000,C 90.000,E1 146.707} C_DIS
LIN {X 0.027,Y -582.598,Z 907.607,A 0.000,B 0.000,C 90.000,E1 145.182} C_DIS
LIN {X -0.145,Y -587.831,Z 907.600,A 0.000,B 0.000,C 90.000,E1 143.989} C_DIS
LIN {X -0.172,Y -592.285,Z 907.594,A 0.000,B 0.000,C 90.000,E1 142.924} C_DIS
LIN {X 0.075,Y -599.829,Z 907.584,A 0.000,B 0.000,C 90.000,E1 141.045} C_DIS
LIN {X 0.160,Y -606.334,Z 907.575,A 0.000,B 0.000,C 90.000,E1 139.461} C_DIS
LIN {X -0.070,Y -612.830,Z 907.566,A 0.000,B 0.000,C 90.000,E1 137.919} C_DIS
LIN {X 0.149,Y -617.281,Z 907.560,A 0.000,B 0.000,C 90.000,E1 136.863} C_DIS
LIN {X 0.112,Y -623.934,Z 907.552,A 0.000,B 0.000,C 90.000,E1 135.324} C_DIS
LIN {X 0.014,Y -628.227,Z 907.546,A 0.000,B 0.000,C 90.000,E1 134.312} C_DIS
LIN {X -0.021,Y -632.458,Z 907.541,A 0.000,B 0.000,C 90.000,E1 133.299} C_DIS
LIN {X 0.004,Y -636.679,Z 907.535,A 0.000,B 0.000,C 90.000,E1 132.285} C_DIS
LIN {X -0.036,Y -642.867,Z 907.527,A 0.000,B 0.000,C 90.000,E1 130.782} C_DIS
LIN {X 0.128,Y -647.686,Z 907.520,A 0.000,B 0.000,C 90.000,E1 129.519} C_DIS
LIN {X -0.068,Y -651.525,Z 907.514,A 0.000,B 0.000,C 90.000,E1 128.543} C_DIS
LIN {X -0.229,Y -657.190,Z 907.506,A 0.000,B 0.000,C 90.000,E1 127.076} C_DIS
LIN {X 0.256,Y -659.876,Z 907.502,A 0.000,B 0.000,C 90.000,E1 126.297} C_DIS
LIN {X 0.390,Y -665.052,Z 907.494,A 0.000,B 0.000,C 90.000,E1 124.818} C_DIS
LIN {X 0.108,Y -669.119,Z 907.487,A 0.000,B 0.000,C 90.000,E1 123.627} C_DIS
LIN {X 0.341,Y -671.328,Z 907.483,A 0.000,B 0.000,C 90.000,E1 122.880} C_DIS
LIN {X -0.331,Y -673.431,Z 907.479,A 0.000,B 0.000,C 90.000,E1 122.212} C_DIS
LIN {X 0.119,Y -675.801,Z 907.474,A 0.000,B 0.000,C 90.000,E1 121.209} C_DIS
LIN {X 0.204,Y -678.378,Z 907.467,A 0.000,B 0.000,C 90.000,E1 120.001} C_DIS
LIN {X -0.211,Y -680.030,Z 907.461,A 0.000,B 0.000,C 90.000,E1 119.077} C_DIS
LIN {X -0.211,Y -681.198,Z 907.458,A 0.000,B 0.000,C 90.000,E1 118.359} C_DIS
LIN {X 0.003,Y -682.406,Z 907.452,A 0.000,B 0.000,C 90.000,E1 117.385} C_DIS
LIN {X 0.138,Y -683.261,Z 907.446,A 0.000,B 0.000,C 90.000,E1 116.181} C_DIS
LIN {X -0.326,Y -683.594,Z 907.439,A 0.000,B 0.000,C 90.000,E1 115.027} C_DIS
LIN {X 0.308,Y -683.508,Z 907.435,A 0.000,B 0.000,C 90.000,E1 114.259} C_DIS
LIN {X -0.177,Y -683.288,Z 907.432,A 0.000,B 0.000,C 90.000,E1 113.823} C_DIS
LIN {X -0.033,Y -682.662,Z 907.430,A 0.000,B 0.000,C 90.000,E1 113.334} C_DIS
LIN {X 0.173,Y -682.235,Z 907.428,A 0.000,B 0.000,C 90.000,E1 113.078} C_DIS
LIN {X -0.216,Y -679.731,Z 907.425,A 0.000,B 0.000,C 90.000,E1 112.514} C_DIS
LIN {X -0.117,Y -679.008,Z 907.424,A 0.000,B 0.000,C 90.000,E1 112.386} C_DIS
LIN {X -0.280,Y -677.909,Z 907.424,A 0.000,B 0.000,C 90.000,E1 112.280} C_DIS
LIN {X 0.141,Y -672.682,Z 907.421,A 0.000,B 0.000,C 90.000,E1 111.791} C_DIS
LIN {X -0.303,Y -670.790,Z 907.421,A 0.000,B 0.000,C 90.000,E1 111.716} C_DIS
LIN {X -0.024,Y -662.126,Z 907.419,A 0.000,B 0.000,C 90.000,E1 111.408} C_DIS
LIN {X -0.057,Y -659.199,Z 907.419,A 0.000,B 0.000,C 90.000,E1 111.354} C_DIS
LIN {X -0.176,Y -656.074,Z 907.418,A 0.000,B 0.000,C 90.000,E1 111.334} C_DIS
LIN {X -0.159,Y -652.963,Z 907.418,A 0.000,B 0.000,C 90.000,E1 111.280} C_DIS
LIN {X -0.072,Y -640.223,Z 907.418,A 0.000,B 0.000,C 90.000,E1 111.153} C_DIS
LIN {X 0.159,Y -633.864,Z 907.417,A 0.000,B 0.000,C 90.000,E1 111.046} C_DIS
LIN {X -0.195,Y -628.008,Z 907.416,A 0.000,B 0.000,C 90.000,E1 110.972} C_DIS
LIN {X -0.174,Y -620.409,Z 907.415,A 0.000,B 0.000,C 90.000,E1 110.791} C_DIS
LIN {X -0.079,Y -613.101,Z 907.414,A 0.000,B 0.000,C 90.000,E1 110.556} C_DIS
LIN {X 0.145,Y -605.944,Z 907.413,A 0.000,B 0.000,C 90.000,E1 110.248} C_DIS
LIN {X -0.078,Y -601.742,Z 907.411,A 0.000,B 0.000,C 90.000,E1 110.066} C_DIS
LIN {X -0.061,Y -596.188,Z 907.410,A 0.000,B 0.000,C 90.000,E1 109.758} C_DIS
LIN {X 0.168,Y -582.574,Z 907.405,A 0.000,B 0.000,C 90.000,E1 108.906} C_DIS
LIN {X -0.257,Y -580.962,Z 907.405,A 0.000,B 0.000,C 90.000,E1 108.852} C_DIS
LIN {X 0.005,Y -572.856,Z 907.402,A 0.000,B 0.000,C 90.000,E1 108.417} C_DIS
LIN {X -0.010,Y -565.517,Z 907.401,A 0.000,B 0.000,C 90.000,E1 108.127} C_DIS
LIN {X -0.073,Y -558.952,Z 907.399,A 0.000,B 0.000,C 90.000,E1 107.873} C_DIS
LIN {X -0.140,Y -556.566,Z 907.399,A 0.000,B 0.000,C 90.000,E1 107.764} C_DIS
LIN {X -0.173,Y -556.531,Z 907.399,A 0.000,B 0.000,C 90.000,E1 107.764} C_DIS
LIN {X -0.171,Y -555.028,Z 907.398,A 0.000,B 0.000,C 90.000,E1 107.583} C_DIS
LIN {X -0.212,Y -555.013,Z 907.398,A 0.000,B 0.000,C 90.000,E1 107.583} C_DIS
LIN {X 0.028,Y -554.552,Z 907.396,A 0.000,B 0.000,C 90.000,E1 107.275} C_DIS
LIN {X 0.130,Y -554.547,Z 907.392,A 0.000,B 0.000,C 90.000,E1 106.567} C_DIS
LIN {X -0.180,Y -555.254,Z 907.381,A 0.000,B 0.000,C 90.000,E1 104.647} C_DIS
LIN {X 0.310,Y -556.277,Z 907.370,A 0.000,B 0.000,C 90.000,E1 102.647} C_DIS
LIN {X -0.209,Y -557.998,Z 907.357,A 0.000,B 0.000,C 90.000,E1 100.197} C_DIS
LIN {X -0.007,Y -559.184,Z 907.347,A 0.000,B 0.000,C 90.000,E1 98.511} C_DIS
LIN {X -0.007,Y -560.142,Z 907.340,A 0.000,B 0.000,C 90.000,E1 97.125} C_DIS
LIN {X 0.093,Y -561.109,Z 907.330,A 0.000,B 0.000,C 90.000,E1 95.454} C_DIS
LIN {X -0.018,Y -561.691,Z 907.324,A 0.000,B 0.000,C 90.000,E1 94.359} C_DIS
LIN {X -0.165,Y -562.224,Z 907.318,A 0.000,B 0.000,C 90.000,E1 93.269} C_DIS
LIN {X -0.201,Y -562.799,Z 907.310,A 0.000,B 0.000,C 90.000,E1 91.892} C_DIS
LIN {X -0.234,Y -563.229,Z 907.303,A 0.000,B 0.000,C 90.000,E1 90.516} C_DIS
LIN {X 0.187,Y -563.566,Z 907.297,A 0.000,B 0.000,C 90.000,E1 89.370} C_DIS
LIN {X 0.274,Y -563.902,Z 907.287,A 0.000,B 0.000,C 90.000,E1 87.707} C_DIS
LIN {X -0.200,Y -564.156,Z 907.278,A 0.000,B 0.000,C 90.000,E1 86.102} C_DIS
LIN {X -0.027,Y -564.475,Z 907.269,A 0.000,B 0.000,C 90.000,E1 84.432} C_DIS
LIN {X 0.000,Y -564.692,Z 907.261,A 0.000,B 0.000,C 90.000,E1 83.053} C_DIS
LIN {X 0.170,Y -565.036,Z 907.254,A 0.000,B 0.000,C 90.000,E1 81.659} C_DIS
LIN {X 0.044,Y -565.678,Z 907.243,A 0.000,B 0.000,C 90.000,E1 79.746} C_DIS
LIN {X -0.152,Y -566.442,Z 907.234,A 0.000,B 0.000,C 90.000,E1 78.117} C_DIS
LIN {X 0.282,Y -567.143,Z 907.226,A 0.000,B 0.000,C 90.000,E1 76.700} C_DIS
LIN {X -0.186,Y -568.054,Z 907.217,A 0.000,B 0.000,C 90.000,E1 75.102} C_DIS
LIN {X -0.266,Y -568.658,Z 907.210,A 0.000,B 0.000,C 90.000,E1 73.740} C_DIS
LIN {X 0.194,Y -569.143,Z 907.203,A 0.000,B 0.000,C 90.000,E1 72.598} C_DIS
LIN {X -0.255,Y -569.652,Z 907.196,A 0.000,B 0.000,C 90.000,E1 71.275} C_DIS
LIN {X 0.022,Y -570.009,Z 907.188,A 0.000,B 0.000,C 90.000,E1 69.880} C_DIS
LIN {X -0.064,Y -570.437,Z 907.178,A 0.000,B 0.000,C 90.000,E1 67.975} C_DIS
LIN {X -0.278,Y -570.648,Z 907.169,A 0.000,B 0.000,C 90.000,E1 66.357} C_DIS
LIN {X 0.090,Y -570.734,Z 907.158,A 0.000,B 0.000,C 90.000,E1 64.409} C_DIS
LIN {X 0.016,Y -570.739,Z 907.150,A 0.000,B 0.000,C 90.000,E1 63.050} C_DIS
LIN {X -0.151,Y -570.750,Z 907.144,A 0.000,B 0.000,C 90.000,E1 61.975} C_DIS
LIN {X -0.014,Y -570.510,Z 907.134,A 0.000,B 0.000,C 90.000,E1 60.049} C_DIS
LIN {X 0.186,Y -570.156,Z 907.126,A 0.000,B 0.000,C 90.000,E1 58.663} C_DIS
LIN {X 0.066,Y -569.767,Z 907.120,A 0.000,B 0.000,C 90.000,E1 57.582} C_DIS
LIN {X -0.136,Y -568.849,Z 907.111,A 0.000,B 0.000,C 90.000,E1 55.960} C_DIS
LIN {X 0.152,Y -567.827,Z 907.103,A 0.000,B 0.000,C 90.000,E1 54.562} C_DIS
LIN {X -0.158,Y -566.727,Z 907.097,A 0.000,B 0.000,C 90.000,E1 53.497} C_DIS
LIN {X -0.139,Y -565.416,Z 907.091,A 0.000,B 0.000,C 90.000,E1 52.396} C_DIS
LIN {X -0.131,Y -563.902,Z 907.085,A 0.000,B 0.000,C 90.000,E1 51.295} C_DIS
LIN {X 0.186,Y -562.592,Z 907.080,A 0.000,B 0.000,C 90.000,E1 50.436} C_DIS
LIN {X -0.284,Y -560.474,Z 907.074,A 0.000,B 0.000,C 90.000,E1 49.380} C_DIS
LIN {X -0.075,Y -558.672,Z 907.070,A 0.000,B 0.000,C 90.000,E1 48.528} C_DIS
LIN {X 0.082,Y -557.341,Z 907.067,A 0.000,B 0.000,C 90.000,E1 47.957} C_DIS
LIN {X 0.188,Y -555.863,Z 907.063,A 0.000,B 0.000,C 90.000,E1 47.391} C_DIS
LIN {X -0.059,Y -553.378,Z 907.059,A 0.000,B 0.000,C 90.000,E1 46.581} C_DIS
LIN {X 0.072,Y -550.574,Z 907.054,A 0.000,B 0.000,C 90.000,E1 45.729} C_DIS
LIN {X -0.224,Y -547.507,Z 907.049,A 0.000,B 0.000,C 90.000,E1 44.919} C_DIS
LIN {X -0.180,Y -545.273,Z 907.046,A 0.000,B 0.000,C 90.000,E1 44.352} C_DIS
LIN {X -0.350,Y -543.533,Z 907.044,A 0.000,B 0.000,C 90.000,E1 43.947} C_DIS
LIN {X -0.143,Y -538.736,Z 907.038,A 0.000,B 0.000,C 90.000,E1 42.933} C_DIS
LIN {X -0.171,Y -535.796,Z 907.035,A 0.000,B 0.000,C 90.000,E1 42.366} C_DIS
LIN {X -0.001,Y -533.462,Z 907.033,A 0.000,B 0.000,C 90.000,E1 41.919} C_DIS
LIN {X -0.255,Y -529.297,Z 907.029,A 0.000,B 0.000,C 90.000,E1 41.229} C_DIS
LIN {X -0.118,Y -526.682,Z 907.027,A 0.000,B 0.000,C 90.000,E1 40.782} C_DIS
LIN {X 0.304,Y -521.993,Z 907.023,A 0.000,B 0.000,C 90.000,E1 40.011} C_DIS
LIN {X -0.060,Y -517.052,Z 907.018,A 0.000,B 0.000,C 90.000,E1 39.322} C_DIS
LIN {X -0.065,Y -511.831,Z 907.014,A 0.000,B 0.000,C 90.000,E1 38.588} C_DIS
LIN {X -0.230,Y -507.269,Z 907.011,A 0.000,B 0.000,C 90.000,E1 38.016} C_DIS
LIN {X -0.023,Y -502.384,Z 907.008,A 0.000,B 0.000,C 90.000,E1 37.397} C_DIS
LIN {X 0.022,Y -496.146,Z 907.004,A 0.000,B 0.000,C 90.000,E1 36.664} C_DIS
LIN {X -0.145,Y -490.734,Z 907.000,A 0.000,B 0.000,C 90.000,E1 36.091} C_DIS
LIN {X -0.158,Y -485.108,Z 906.997,A 0.000,B 0.000,C 90.000,E1 35.518} C_DIS
LIN {X 0.140,Y -476.750,Z 906.993,A 0.000,B 0.000,C 90.000,E1 34.692} C_DIS
LIN {X -0.032,Y -467.827,Z 906.988,A 0.000,B 0.000,C 90.000,E1 33.913} C_DIS
LIN {X 0.074,Y -458.681,Z 906.984,A 0.000,B 0.000,C 90.000,E1 33.118} C_DIS
LIN {X 0.144,Y -449.472,Z 906.980,A 0.000,B 0.000,C 90.000,E1 32.339} C_DIS
LIN {X 0.042,Y -435.562,Z 906.973,A 0.000,B 0.000,C 90.000,E1 31.209} C_DIS
LIN {X 0.022,Y -421.911,Z 906.967,A 0.000,B 0.000,C 90.000,E1 30.050} C_DIS
LIN {X 0.172,Y -405.380,Z 906.958,A 0.000,B 0.000,C 90.000,E1 28.487} C_DIS
LIN {X 0.120,Y -399.571,Z 906.955,A 0.000,B 0.000,C 90.000,E1 27.897} C_DIS
LIN {X -0.107,Y -396.009,Z 906.953,A 0.000,B 0.000,C 90.000,E1 27.513} C_DIS
LIN {X 0.195,Y -393.493,Z 906.951,A 0.000,B 0.000,C 90.000,E1 27.129} C_DIS
LIN {X -0.137,Y -392.405,Z 906.950,A 0.000,B 0.000,C 90.000,E1 27.001} C_DIS
LIN {X -0.046,Y -390.670,Z 906.948,A 0.000,B 0.000,C 90.000,E1 26.616} C_DIS
LIN {X -0.188,Y -389.395,Z 906.945,A 0.000,B 0.000,C 90.000,E1 26.104} C_DIS
LIN {X 0.219,Y -388.844,Z 906.941,A 0.000,B 0.000,C 90.000,E1 25.335} C_DIS
LIN {X 0.014,Y -388.909,Z 906.937,A 0.000,B 0.000,C 90.000,E1 24.591} C_DIS
LIN {X 0.081,Y -389.774,Z 906.929,A 0.000,B 0.000,C 90.000,E1 23.153} C_DIS
LIN {X -0.158,Y -393.238,Z 906.909,A 0.000,B 0.000,C 90.000,E1 19.631} C_DIS
LIN {X -0.182,Y -396.536,Z 906.893,A 0.000,B 0.000,C 90.000,E1 16.804} C_DIS
LIN {X 0.094,Y -399.631,Z 906.880,A 0.000,B 0.000,C 90.000,E1 14.300} C_DIS
LIN {X -0.214,Y -402.537,Z 906.868,A 0.000,B 0.000,C 90.000,E1 12.243} C_DIS
LIN {X -0.129,Y -406.247,Z 906.854,A 0.000,B 0.000,C 90.000,E1 9.792} C_DIS
LIN {X -0.012,Y -411.530,Z 906.837,A 0.000,B 0.000,C 90.000,E1 6.663} C_DIS
LIN {X 0.142,Y -416.688,Z 906.822,A 0.000,B 0.000,C 90.000,E1 3.898} C_DIS
LIN {X -0.042,Y -422.490,Z 906.807,A 0.000,B 0.000,C 90.000,E1 1.203} C_DIS
LIN {X 0.119,Y -430.826,Z 906.788,A 0.000,B 0.000,C 90.000,E1 357.764} C_DIS
LIN {X -0.165,Y -432.722,Z 906.784,A 0.000,B 0.000,C 90.000,E1 357.135} C_DIS
LIN {X -0.022,Y -434.486,Z 906.781,A 0.000,B 0.000,C 90.000,E1 356.617} C_DIS
LIN {X 0.056,Y -436.528,Z 906.779,A 0.000,B 0.000,C 90.000,E1 356.159} C_DIS
LIN {X 0.102,Y -437.574,Z 906.778,A 0.000,B 0.000,C 90.000,E1 355.988} C_DIS
LIN {X -0.172,Y -440.777,Z 906.776,A 0.000,B 0.000,C 90.000,E1 355.641} C_DIS
LIN {X -0.081,Y -442.390,Z 906.775,A 0.000,B 0.000,C 90.000,E1 355.469} C_DIS
LIN {X 0.160,Y -447.975,Z 906.773,A 0.000,B 0.000,C 90.000,E1 355.065} C_DIS
LIN {X -0.216,Y -462.872,Z 906.769,A 0.000,B 0.000,C 90.000,E1 354.432} C_DIS
LIN {X 0.022,Y -473.099,Z 906.766,A 0.000,B 0.000,C 90.000,E1 353.913} C_DIS
LIN {X 0.148,Y -483.078,Z 906.763,A 0.000,B 0.000,C 90.000,E1 353.394} C_DIS
LIN {X 0.190,Y -494.559,Z 906.760,A 0.000,B 0.000,C 90.000,E1 352.761} C_DIS
LIN {X 0.079,Y -506.087,Z 906.756,A 0.000,B 0.000,C 90.000,E1 352.129} C_DIS
LIN {X 0.059,Y -515.441,Z 906.753,A 0.000,B 0.000,C 90.000,E1 351.546} C_DIS
LIN {X 0.158,Y -524.764,Z 906.750,A 0.000,B 0.000,C 90.000,E1 350.914} C_DIS
LIN {X 0.030,Y -530.855,Z 906.747,A 0.000,B 0.000,C 90.000,E1 350.500} C_DIS
LIN {X 0.070,Y -538.130,Z 906.744,A 0.000,B 0.000,C 90.000,E1 349.926} C_DIS
LIN {X -0.163,Y -545.164,Z 906.741,A 0.000,B 0.000,C 90.000,E1 349.342} C_DIS
LIN {X -0.087,Y -551.792,Z 906.737,A 0.000,B 0.000,C 90.000,E1 348.701} C_DIS
LIN {X -0.179,Y -558.144,Z 906.734,A 0.000,B 0.000,C 90.000,E1 348.049} C_DIS
LIN {X -0.180,Y -562.922,Z 906.731,A 0.000,B 0.000,C 90.000,E1 347.521} C_DIS
LIN {X -0.241,Y -569.902,Z 906.726,A 0.000,B 0.000,C 90.000,E1 346.700} C_DIS
LIN {X 0.128,Y -574.120,Z 906.723,A 0.000,B 0.000,C 90.000,E1 346.117} C_DIS
LIN {X 0.324,Y -580.127,Z 906.718,A 0.000,B 0.000,C 90.000,E1 345.283} C_DIS
LIN {X -0.216,Y -586.502,Z 906.713,A 0.000,B 0.000,C 90.000,E1 344.393} C_DIS
LIN {X 0.188,Y -590.720,Z 906.710,A 0.000,B 0.000,C 90.000,E1 343.685} C_DIS
LIN {X -0.132,Y -596.930,Z 906.704,A 0.000,B 0.000,C 90.000,E1 342.653} C_DIS
LIN {X -0.023,Y -603.344,Z 906.697,A 0.000,B 0.000,C 90.000,E1 341.456} C_DIS
LIN {X -0.166,Y -608.681,Z 906.691,A 0.000,B 0.000,C 90.000,E1 340.423} C_DIS
LIN {X -0.218,Y -613.152,Z 906.686,A 0.000,B 0.000,C 90.000,E1 339.518} C_DIS
LIN {X -0.015,Y -617.976,Z 906.680,A 0.000,B 0.000,C 90.000,E1 338.465} C_DIS
LIN {X 0.253,Y -622.558,Z 906.675,A 0.000,B 0.000,C 90.000,E1 337.411} C_DIS
LIN {X -0.231,Y -627.747,Z 906.668,A 0.000,B 0.000,C 90.000,E1 336.177} C_DIS
LIN {X -0.121,Y -632.453,Z 906.661,A 0.000,B 0.000,C 90.000,E1 334.897} C_DIS
LIN {X -0.197,Y -636.964,Z 906.654,A 0.000,B 0.000,C 90.000,E1 333.640} C_DIS
LIN {X 0.015,Y -640.196,Z 906.648,A 0.000,B 0.000,C 90.000,E1 332.615} C_DIS
LIN {X -0.300,Y -643.191,Z 906.642,A 0.000,B 0.000,C 90.000,E1 331.641} C_DIS
LIN {X -0.186,Y -646.624,Z 906.635,A 0.000,B 0.000,C 90.000,E1 330.383} C_DIS
LIN {X -0.093,Y -649.243,Z 906.630,A 0.000,B 0.000,C 90.000,E1 329.380} C_DIS
LIN {X -0.306,Y -651.726,Z 906.624,A 0.000,B 0.000,C 90.000,E1 328.408} C_DIS
LIN {X 0.195,Y -653.982,Z 906.619,A 0.000,B 0.000,C 90.000,E1 327.375} C_DIS
LIN {X -0.174,Y -655.904,Z 906.613,A 0.000,B 0.000,C 90.000,E1 326.421} C_DIS
LIN {X 0.388,Y -657.595,Z 906.608,A 0.000,B 0.000,C 90.000,E1 325.388} C_DIS
LIN {X 0.050,Y -659.015,Z 906.602,A 0.000,B 0.000,C 90.000,E1 324.436} C_DIS
LIN {X 0.051,Y -660.554,Z 906.596,A 0.000,B 0.000,C 90.000,E1 323.210} C_DIS
LIN {X 0.083,Y -661.816,Z 906.589,A 0.000,B 0.000,C 90.000,E1 321.984} C_DIS
LIN {X -0.384,Y -662.964,Z 906.582,A 0.000,B 0.000,C 90.000,E1 320.803} C_DIS
LIN {X 0.100,Y -664.115,Z 906.575,A 0.000,B 0.000,C 90.000,E1 319.542} C_DIS
LIN {X 0.077,Y -666.027,Z 906.565,A 0.000,B 0.000,C 90.000,E1 317.595} C_DIS
LIN {X 0.102,Y -667.024,Z 906.559,A 0.000,B 0.000,C 90.000,E1 316.620} C_DIS
LIN {X 0.110,Y -667.937,Z 906.554,A 0.000,B 0.000,C 90.000,E1 315.648} C_DIS
LIN {X 0.150,Y -669.262,Z 906.546,A 0.000,B 0.000,C 90.000,E1 314.190} C_DIS
LIN {X -0.243,Y -670.804,Z 906.536,A 0.000,B 0.000,C 90.000,E1 312.528} C_DIS
LIN {X -0.134,Y -671.948,Z 906.529,A 0.000,B 0.000,C 90.000,E1 311.310} C_DIS
LIN {X -0.007,Y -672.904,Z 906.523,A 0.000,B 0.000,C 90.000,E1 310.092} C_DIS
LIN {X 0.235,Y -674.063,Z 906.515,A 0.000,B 0.000,C 90.000,E1 308.624} C_DIS
LIN {X -0.039,Y -675.028,Z 906.508,A 0.000,B 0.000,C 90.000,E1 307.443} C_DIS
LIN {X 0.230,Y -675.776,Z 906.501,A 0.000,B 0.000,C 90.000,E1 306.217} C_DIS
LIN {X -0.290,Y -676.536,Z 906.493,A 0.000,B 0.000,C 90.000,E1 304.818} C_DIS
LIN {X -0.088,Y -677.508,Z 906.483,A 0.000,B 0.000,C 90.000,E1 302.880} C_DIS
LIN {X -0.197,Y -678.658,Z 906.473,A 0.000,B 0.000,C 90.000,E1 301.209} C_DIS
LIN {X -0.072,Y -681.014,Z 906.459,A 0.000,B 0.000,C 90.000,E1 298.565} C_DIS
LIN {X 0.164,Y -683.062,Z 906.449,A 0.000,B 0.000,C 90.000,E1 296.873} C_DIS
LIN {X 0.056,Y -685.694,Z 906.439,A 0.000,B 0.000,C 90.000,E1 294.975} C_DIS
LIN {X 0.031,Y -686.837,Z 906.434,A 0.000,B 0.000,C 90.000,E1 294.027} C_DIS
LIN {X -0.157,Y -687.324,Z 906.431,A 0.000,B 0.000,C 90.000,E1 293.567} C_DIS
LIN {X 0.012,Y -687.529,Z 906.428,A 0.000,B 0.000,C 90.000,E1 293.078} C_DIS
LIN {X 0.232,Y -687.489,Z 906.427,A 0.000,B 0.000,C 90.000,E1 292.823} C_DIS
LIN {X -0.229,Y -686.844,Z 906.424,A 0.000,B 0.000,C 90.000,E1 292.386} C_DIS
LIN {X -0.272,Y -686.155,Z 906.423,A 0.000,B 0.000,C 90.000,E1 292.153} C_DIS
LIN {X -0.057,Y -684.919,Z 906.422,A 0.000,B 0.000,C 90.000,E1 291.897} C_DIS
LIN {X 0.002,Y -682.556,Z 906.420,A 0.000,B 0.000,C 90.000,E1 291.535} C_DIS
LIN {X 0.103,Y -681.416,Z 906.419,A 0.000,B 0.000,C 90.000,E1 291.408} C_DIS
LIN {X 0.200,Y -679.662,Z 906.418,A 0.000,B 0.000,C 90.000,E1 291.280} C_DIS
LIN {X -0.263,Y -674.185,Z 906.417,A 0.000,B 0.000,C 90.000,E1 291.046} C_DIS
LIN {X 0.241,Y -672.609,Z 906.416,A 0.000,B 0.000,C 90.000,E1 290.918} C_DIS
LIN {X -0.107,Y -664.628,Z 906.414,A 0.000,B 0.000,C 90.000,E1 290.610} C_DIS
LIN {X -0.269,Y -660.859,Z 906.413,A 0.000,B 0.000,C 90.000,E1 290.429} C_DIS
LIN {X -0.328,Y -660.800,Z 906.413,A 0.000,B 0.000,C 90.000,E1 290.429} C_DIS
LIN {X 0.252,Y -660.277,Z 906.413,A 0.000,B 0.000,C 90.000,E1 290.301} C_DIS
LIN {X 0.192,Y -660.257,Z 906.413,A 0.000,B 0.000,C 90.000,E1 290.301} C_DIS
LIN {X 0.076,Y -660.284,Z 906.412,A 0.000,B 0.000,C 90.000,E1 290.066} C_DIS
LIN {X 0.101,Y -661.996,Z 906.409,A 0.000,B 0.000,C 90.000,E1 289.523} C_DIS
LIN {X 0.168,Y -664.713,Z 906.405,A 0.000,B 0.000,C 90.000,E1 288.906} C_DIS
LIN {X 0.154,Y -671.060,Z 906.398,A 0.000,B 0.000,C 90.000,E1 287.692} C_DIS
LIN {X -0.053,Y -674.401,Z 906.394,A 0.000,B 0.000,C 90.000,E1 286.985} C_DIS
LIN {X 0.023,Y -676.359,Z 906.392,A 0.000,B 0.000,C 90.000,E1 286.496} C_DIS
LIN {X -0.126,Y -678.782,Z 906.388,A 0.000,B 0.000,C 90.000,E1 285.788} C_DIS
LIN {X -0.072,Y -680.661,Z 906.384,A 0.000,B 0.000,C 90.000,E1 285.064} C_DIS
LIN {X -0.211,Y -682.726,Z 906.378,A 0.000,B 0.000,C 90.000,E1 284.120} C_DIS
LIN {X -0.298,Y -683.984,Z 906.374,A 0.000,B 0.000,C 90.000,E1 283.411} C_DIS
LIN {X 0.269,Y -685.268,Z 906.369,A 0.000,B 0.000,C 90.000,E1 282.411} C_DIS
LIN {X 0.060,Y -685.922,Z 906.365,A 0.000,B 0.000,C 90.000,E1 281.715} C_DIS
LIN {X 0.018,Y -686.143,Z 906.362,A 0.000,B 0.000,C 90.000,E1 281.243} C_DIS
LIN {X -0.155,Y -686.107,Z 906.360,A 0.000,B 0.000,C 90.000,E1 280.782} C_DIS
LIN {X -0.200,Y -685.752,Z 906.357,A 0.000,B 0.000,C 90.000,E1 280.310} C_DIS
LIN {X -0.224,Y -685.460,Z 906.356,A 0.000,B 0.000,C 90.000,E1 280.074} C_DIS
LIN {X 0.280,Y -684.583,Z 906.353,A 0.000,B 0.000,C 90.000,E1 279.557} C_DIS
LIN {X 0.108,Y -683.374,Z 906.351,A 0.000,B 0.000,C 90.000,E1 279.095} C_DIS
LIN {X 0.035,Y -681.753,Z 906.348,A 0.000,B 0.000,C 90.000,E1 278.624} C_DIS
LIN {X -0.107,Y -680.869,Z 906.347,A 0.000,B 0.000,C 90.000,E1 278.398} C_DIS
LIN {X -0.295,Y -678.787,Z 906.344,A 0.000,B 0.000,C 90.000,E1 277.936} C_DIS
LIN {X 0.115,Y -675.264,Z 906.340,A 0.000,B 0.000,C 90.000,E1 277.182} C_DIS
LIN {X -0.111,Y -672.684,Z 906.337,A 0.000,B 0.000,C 90.000,E1 276.720} C_DIS
LIN {X 0.313,Y -669.872,Z 906.335,A 0.000,B 0.000,C 90.000,E1 276.201} C_DIS
LIN {X 0.052,Y -666.820,Z 906.332,A 0.000,B 0.000,C 90.000,E1 275.739} C_DIS
LIN {X -0.317,Y -662.463,Z 906.329,A 0.000,B 0.000,C 90.000,E1 275.163} C_DIS
LIN {X 0.031,Y -658.607,Z 906.326,A 0.000,B 0.000,C 90.000,E1 274.645} C_DIS
LIN {X 0.301,Y -654.333,Z 906.323,A 0.000,B 0.000,C 90.000,E1 274.131} C_DIS
LIN {X -0.060,Y -649.662,Z 906.320,A 0.000,B 0.000,C 90.000,E1 273.669} C_DIS
LIN {X -0.336,Y -644.635,Z 906.318,A 0.000,B 0.000,C 90.000,E1 273.212} C_DIS
LIN {X 0.302,Y -637.929,Z 906.315,A 0.000,B 0.000,C 90.000,E1 272.579} C_DIS
LIN {X -0.090,Y -630.721,Z 906.311,A 0.000,B 0.000,C 90.000,E1 272.064} C_DIS
LIN {X 0.033,Y -623.148,Z 906.309,A 0.000,B 0.000,C 90.000,E1 271.547} C_DIS
LIN {X 0.243,Y -616.898,Z 906.307,A 0.000,B 0.000,C 90.000,E1 271.146} C_DIS
LIN {X -0.155,Y -608.473,Z 906.304,A 0.000,B 0.000,C 90.000,E1 270.745} C_DIS
LIN {X 0.278,Y -603.434,Z 906.303,A 0.000,B 0.000,C 90.000,E1 270.458} C_DIS
LIN {X 0.043,Y -596.539,Z 906.301,A 0.000,B 0.000,C 90.000,E1 270.172} C_DIS
LIN {X 0.268,Y -591.180,Z 906.300,A 0.000,B 0.000,C 90.000,E1 269.943} C_DIS
LIN {X 0.085,Y -583.896,Z 906.299,A 0.000,B 0.000,C 90.000,E1 269.714} C_DIS
LIN {X 0.276,Y -578.632,Z 906.298,A 0.000,B 0.000,C 90.000,E1 269.542} C_DIS
LIN {X -0.014,Y -572.390,Z 906.297,A 0.000,B 0.000,C 90.000,E1 269.427} C_DIS
LIN {X -0.197,Y -567.978,Z 906.296,A 0.000,B 0.000,C 90.000,E1 269.370} C_DIS
LIN {X -0.260,Y -563.416,Z 906.296,A 0.000,B 0.000,C 90.000,E1 269.312} C_DIS
LIN {X 0.039,Y -553.047,Z 906.296,A 0.000,B 0.000,C 90.000,E1 269.198} C_DIS
LIN {X -0.049,Y -550.336,Z 906.295,A 0.000,B 0.000,C 90.000,E1 269.141} C_DIS
LIN {X -0.202,Y -549.784,Z 906.295,A 0.000,B 0.000,C 90.000,E1 269.141} C_DIS
LIN {X -0.232,Y -549.719,Z 906.295,A 0.000,B 0.000,C 90.000,E1 269.141} C_DIS
LIN {X 0.236,Y -547.670,Z 906.294,A 0.000,B 0.000,C 90.000,E1 268.912} C_DIS
LIN {X 0.195,Y -545.403,Z 906.293,A 0.000,B 0.000,C 90.000,E1 268.682} C_DIS
LIN {X 0.139,Y -545.373,Z 906.293,A 0.000,B 0.000,C 90.000,E1 268.682} C_DIS
LIN {X 0.058,Y -544.181,Z 906.291,A 0.000,B 0.000,C 90.000,E1 268.339} C_DIS
LIN {X -0.264,Y -543.208,Z 906.287,A 0.000,B 0.000,C 90.000,E1 267.650} C_DIS
LIN {X 0.135,Y -540.343,Z 906.268,A 0.000,B 0.000,C 90.000,E1 264.204} C_DIS
LIN {X -0.267,Y -539.535,Z 906.262,A 0.000,B 0.000,C 90.000,E1 263.109} C_DIS
LIN {X -0.079,Y -538.593,Z 906.255,A 0.000,B 0.000,C 90.000,E1 261.951} C_DIS
LIN {X 0.162,Y -537.253,Z 906.247,A 0.000,B 0.000,C 90.000,E1 260.500} C_DIS
LIN {X -0.213,Y -536.069,Z 906.241,A 0.000,B 0.000,C 90.000,E1 259.398} C_DIS
LIN {X 0.018,Y -534.830,Z 906.235,A 0.000,B 0.000,C 90.000,E1 258.229} C_DIS
LIN {X -0.246,Y -533.201,Z 906.227,A 0.000,B 0.000,C 90.000,E1 256.825} C_DIS
LIN {X 0.267,Y -531.059,Z 906.217,A 0.000,B 0.000,C 90.000,E1 255.046} C_DIS
LIN {X -0.266,Y -528.534,Z 906.206,A 0.000,B 0.000,C 90.000,E1 253.087} C_DIS
LIN {X -0.225,Y -526.781,Z 906.198,A 0.000,B 0.000,C 90.000,E1 251.638} C_DIS
LIN {X -0.051,Y -524.556,Z 906.188,A 0.000,B 0.000,C 90.000,E1 249.880} C_DIS
LIN {X 0.090,Y -522.551,Z 906.180,A 0.000,B 0.000,C 90.000,E1 248.411} C_DIS
LIN {X 0.234,Y -520.972,Z 906.174,A 0.000,B 0.000,C 90.000,E1 247.230} C_DIS
LIN {X -0.122,Y -519.320,Z 906.167,A 0.000,B 0.000,C 90.000,E1 246.102} C_DIS
LIN {X 0.121,Y -516.264,Z 906.156,A 0.000,B 0.000,C 90.000,E1 244.024} C_DIS
LIN {X -0.081,Y -514.390,Z 906.149,A 0.000,B 0.000,C 90.000,E1 242.871} C_DIS
LIN {X 0.030,Y -511.884,Z 906.141,A 0.000,B 0.000,C 90.000,E1 241.385} C_DIS
LIN {X -0.133,Y -508.174,Z 906.130,A 0.000,B 0.000,C 90.000,E1 239.331} C_DIS
LIN {X 0.043,Y -506.080,Z 906.123,A 0.000,B 0.000,C 90.000,E1 238.122} C_DIS
LIN {X 0.184,Y -503.813,Z 906.116,A 0.000,B 0.000,C 90.000,E1 236.914} C_DIS
LIN {X 0.261,Y -501.949,Z 906.111,A 0.000,B 0.000,C 90.000,E1 236.008} C_DIS
LIN {X -0.257,Y -500.683,Z 906.108,A 0.000,B 0.000,C 90.000,E1 235.468} C_DIS
LIN {X -0.037,Y -495.813,Z 906.096,A 0.000,B 0.000,C 90.000,E1 233.336} C_DIS
LIN {X -0.041,Y -492.467,Z 906.088,A 0.000,B 0.000,C 90.000,E1 231.823} C_DIS
LIN {X -0.133,Y -487.715,Z 906.076,A 0.000,B 0.000,C 90.000,E1 229.703} C_DIS
LIN {X -0.187,Y -485.041,Z 906.069,A 0.000,B 0.000,C 90.000,E1 228.485} C_DIS
LIN {X 0.230,Y -479.508,Z 906.056,A 0.000,B 0.000,C 90.000,E1 225.972} C_DIS
LIN {X 0.144,Y -476.021,Z 906.047,A 0.000,B 0.000,C 90.000,E1 224.433} C_DIS
LIN {X -0.238,Y -471.719,Z 906.037,A 0.000,B 0.000,C 90.000,E1 222.609} C_DIS
LIN {X 0.044,Y -466.842,Z 906.024,A 0.000,B 0.000,C 90.000,E1 220.378} C_DIS
LIN {X -0.208,Y -463.456,Z 906.016,A 0.000,B 0.000,C 90.000,E1 218.830} C_DIS
LIN {X -0.156,Y -460.111,Z 906.007,A 0.000,B 0.000,C 90.000,E1 217.237} C_DIS
LIN {X 0.197,Y -456.785,Z 905.998,A 0.000,B 0.000,C 90.000,E1 215.598} C_DIS
LIN {X 0.216,Y -453.339,Z 905.989,A 0.000,B 0.000,C 90.000,E1 213.992} C_DIS
LIN {X 0.082,Y -448.307,Z 905.977,A 0.000,B 0.000,C 90.000,E1 211.750} C_DIS
LIN {X -0.003,Y -445.471,Z 905.969,A 0.000,B 0.000,C 90.000,E1 210.463} C_DIS
LIN {X 0.130,Y -441.258,Z 905.958,A 0.000,B 0.000,C 90.000,E1 208.487} C_DIS
LIN {X -0.052,Y -436.870,Z 905.947,A 0.000,B 0.000,C 90.000,E1 206.539} C_DIS
LIN {X 0.247,Y -432.567,Z 905.936,A 0.000,B 0.000,C 90.000,E1 204.515} C_DIS
LIN {X 0.264,Y -428.220,Z 905.925,A 0.000,B 0.000,C 90.000,E1 202.514} C_DIS
LIN {X 0.067,Y -424.661,Z 905.916,A 0.000,B 0.000,C 90.000,E1 200.865} C_DIS
LIN {X -0.189,Y -421.152,Z 905.907,A 0.000,B 0.000,C 90.000,E1 199.214} C_DIS
LIN {X -0.125,Y -417.764,Z 905.897,A 0.000,B 0.000,C 90.000,E1 197.511} C_DIS
LIN {X 0.160,Y -413.656,Z 905.886,A 0.000,B 0.000,C 90.000,E1 195.426} C_DIS
LIN {X 0.118,Y -410.165,Z 905.876,A 0.000,B 0.000,C 90.000,E1 193.716} C_DIS
LIN {X 0.010,Y -406.855,Z 905.867,A 0.000,B 0.000,C 90.000,E1 192.007} C_DIS
LIN {X 0.142,Y -403.464,Z 905.857,A 0.000,B 0.000,C 90.000,E1 190.254} C_DIS
LIN {X 0.118,Y -399.227,Z 905.846,A 0.000,B 0.000,C 90.000,E1 188.163} C_DIS
LIN {X -0.114,Y -395.055,Z 905.834,A 0.000,B 0.000,C 90.000,E1 186.087} C_DIS
LIN {X -0.053,Y -391.281,Z 905.822,A 0.000,B 0.000,C 90.000,E1 183.955} C_DIS
LIN {X 0.144,Y -387.189,Z 905.808,A 0.000,B 0.000,C 90.000,E1 181.432} C_DIS
LIN {X 0.138,Y -384.871,Z 905.800,A 0.000,B 0.000,C 90.000,E1 180.000} C_DIS
LIN {X -0.120,Y -381.550,Z 905.788,A 0.000,B 0.000,C 90.000,E1 177.879} C_DIS
LIN {X 0.076,Y -377.588,Z 905.772,A 0.000,B 0.000,C 90.000,E1 174.951} C_DIS
LIN {X -0.159,Y -376.542,Z 905.762,A 0.000,B 0.000,C 90.000,E1 173.166} C_DIS
LIN {X 0.084,Y -376.863,Z 905.758,A 0.000,B 0.000,C 90.000,E1 172.413} C_DIS
LIN {X -0.021,Y -377.258,Z 905.756,A 0.000,B 0.000,C 90.000,E1 172.064} C_DIS
LIN {X -0.180,Y -377.863,Z 905.754,A 0.000,B 0.000,C 90.000,E1 171.724} C_DIS
LIN {X 0.095,Y -379.608,Z 905.750,A 0.000,B 0.000,C 90.000,E1 170.971} C_DIS
LIN {X -0.011,Y -381.657,Z 905.747,A 0.000,B 0.000,C 90.000,E1 170.443} C_DIS
LIN {X -0.100,Y -383.539,Z 905.745,A 0.000,B 0.000,C 90.000,E1 170.095} C_DIS
LIN {X -0.177,Y -384.659,Z 905.744,A 0.000,B 0.000,C 90.000,E1 169.926} C_DIS
LIN {X 0.124,Y -387.891,Z 905.742,A 0.000,B 0.000,C 90.000,E1 169.454} C_DIS
LIN {X 0.209,Y -393.340,Z 905.739,A 0.000,B 0.000,C 90.000,E1 168.926} C_DIS
LIN {X 0.196,Y -401.631,Z 905.735,A 0.000,B 0.000,C 90.000,E1 168.342} C_DIS
LIN {X -0.168,Y -409.781,Z 905.733,A 0.000,B 0.000,C 90.000,E1 167.881} C_DIS
LIN {X -0.169,Y -421.298,Z 905.728,A 0.000,B 0.000,C 90.000,E1 167.117} C_DIS
LIN {X 0.069,Y -429.277,Z 905.725,A 0.000,B 0.000,C 90.000,E1 166.520} C_DIS
LIN {X -0.082,Y -437.131,Z 905.722,A 0.000,B 0.000,C 90.000,E1 165.936} C_DIS
LIN {X 0.190,Y -449.191,Z 905.716,A 0.000,B 0.000,C 90.000,E1 164.866} C_DIS
LIN {X 0.082,Y -456.439,Z 905.712,A 0.000,B 0.000,C 90.000,E1 164.212} C_DIS
LIN {X 0.114,Y -460.746,Z 905.710,A 0.000,B 0.000,C 90.000,E1 163.795} C_DIS
LIN {X -0.143,Y -469.095,Z 905.705,A 0.000,B 0.000,C 90.000,E1 162.960} C_DIS
LIN {X -0.011,Y -477.284,Z 905.700,A 0.000,B 0.000,C 90.000,E1 162.054} C_DIS
LIN {X -0.078,Y -482.533,Z 905.697,A 0.000,B 0.000,C 90.000,E1 161.456} C_DIS
LIN {X -0.138,Y -487.433,Z 905.694,A 0.000,B 0.000,C 90.000,E1 160.859} C_DIS
LIN {X 0.145,Y -492.223,Z 905.690,A 0.000,B 0.000,C 90.000,E1 160.242} C_DIS
LIN {X -0.235,Y -503.379,Z 905.682,A 0.000,B 0.000,C 90.000,E1 158.773} C_DIS
LIN {X 0.214,Y -508.706,Z 905.678,A 0.000,B 0.000,C 90.000,E1 157.975} C_DIS
LIN {X -0.156,Y -518.716,Z 905.670,A 0.000,B 0.000,C 90.000,E1 156.538} C_DIS
LIN {X -0.197,Y -524.674,Z 905.665,A 0.000,B 0.000,C 90.000,E1 155.665} C_DIS
LIN {X 0.082,Y -533.097,Z 905.657,A 0.000,B 0.000,C 90.000,E1 154.332} C_DIS
LIN {X -0.109,Y -541.927,Z 905.650,A 0.000,B 0.000,C 90.000,E1 152.922} C_DIS
LIN {X 0.089,Y -548.383,Z 905.643,A 0.000,B 0.000,C 90.000,E1 151.769} C_DIS
LIN {X 0.197,Y -557.496,Z 905.634,A 0.000,B 0.000,C 90.000,E1 150.078} C_DIS
LIN {X -0.294,Y -566.570,Z 905.624,A 0.000,B 0.000,C 90.000,E1 148.329} C_DIS
LIN {X 0.124,Y -571.280,Z 905.619,A 0.000,B 0.000,C 90.000,E1 147.327} C_DIS
LIN {X 0.205,Y -575.133,Z 905.614,A 0.000,B 0.000,C 90.000,E1 146.501} C_DIS
LIN {X 0.011,Y -580.071,Z 905.608,A 0.000,B 0.000,C 90.000,E1 145.435} C_DIS
LIN {X 0.208,Y -585.998,Z 905.601,A 0.000,B 0.000,C 90.000,E1 144.069} C_DIS
LIN {X -0.043,Y -589.495,Z 905.596,A 0.000,B 0.000,C 90.000,E1 143.290} C_DIS
LIN {X -0.102,Y -598.234,Z 905.584,A 0.000,B 0.000,C 90.000,E1 141.170} C_DIS
LIN {X -0.044,Y -604.812,Z 905.576,A 0.000,B 0.000,C 90.000,E1 139.585} C_DIS
LIN {X 0.075,Y -614.683,Z 905.563,A 0.000,B 0.000,C 90.000,E1 137.229} C_DIS
LIN {X 0.290,Y -622.519,Z 905.552,A 0.000,B 0.000,C 90.000,E1 135.405} C_DIS
LIN {X 0.368,Y -629.024,Z 905.544,A 0.000,B 0.000,C 90.000,E1 133.866} C_DIS
LIN {X 0.240,Y -634.313,Z 905.537,A 0.000,B 0.000,C 90.000,E1 132.609} C_DIS
LIN {X -0.325,Y -640.559,Z 905.529,A 0.000,B 0.000,C 90.000,E1 131.148} C_DIS
LIN {X -0.023,Y -642.651,Z 905.526,A 0.000,B 0.000,C 90.000,E1 130.620} C_DIS
LIN {X -0.022,Y -649.358,Z 905.516,A 0.000,B 0.000,C 90.000,E1 128.874} C_DIS
LIN {X 0.284,Y -655.022,Z 905.508,A 0.000,B 0.000,C 90.000,E1 127.363} C_DIS
LIN {X -0.174,Y -657.803,Z 905.504,A 0.000,B 0.000,C 90.000,E1 126.664} C_DIS
LIN {X -0.135,Y -663.895,Z 905.494,A 0.000,B 0.000,C 90.000,E1 124.945} C_DIS
LIN {X 0.115,Y -667.964,Z 905.487,A 0.000,B 0.000,C 90.000,E1 123.706} C_DIS
LIN {X 0.337,Y -670.230,Z 905.483,A 0.000,B 0.000,C 90.000,E1 122.959} C_DIS
LIN {X 0.174,Y -672.989,Z 905.478,A 0.000,B 0.000,C 90.000,E1 122.005} C_DIS
LIN {X 0.097,Y -674.733,Z 905.474,A 0.000,B 0.000,C 90.000,E1 121.288} C_DIS
LIN {X 0.169,Y -677.327,Z 905.467,A 0.000,B 0.000,C 90.000,E1 120.079} C_DIS
LIN {X -0.045,Y -678.216,Z 905.465,A 0.000,B 0.000,C 90.000,E1 119.617} C_DIS
LIN {X -0.133,Y -679.777,Z 905.459,A 0.000,B 0.000,C 90.000,E1 118.665} C_DIS
LIN {X 0.260,Y -680.528,Z 905.457,A 0.000,B 0.000,C 90.000,E1 118.153} C_DIS
LIN {X 0.151,Y -681.683,Z 905.451,A 0.000,B 0.000,C 90.000,E1 117.206} C_DIS
LIN {X 0.373,Y -682.402,Z 905.446,A 0.000,B 0.000,C 90.000,E1 116.232} C_DIS
LIN {X -0.111,Y -682.756,Z 905.439,A 0.000,B 0.000,C 90.000,E1 115.079} C_DIS
LIN {X 0.230,Y -682.746,Z 905.435,A 0.000,B 0.000,C 90.000,E1 114.335} C_DIS
LIN {X -0.256,Y -682.540,Z 905.433,A 0.000,B 0.000,C 90.000,E1 113.898} C_DIS
LIN {X -0.049,Y -682.330,Z 905.431,A 0.000,B 0.000,C 90.000,E1 113.643} C_DIS
LIN {X 0.091,Y -681.626,Z 905.429,A 0.000,B 0.000,C 90.000,E1 113.153} C_DIS
LIN {X 0.293,Y -680.812,Z 905.427,A 0.000,B 0.000,C 90.000,E1 112.898} C_DIS
LIN {X -0.200,Y -678.705,Z 905.425,A 0.000,B 0.000,C 90.000,E1 112.461} C_DIS
LIN {X -0.105,Y -677.766,Z 905.424,A 0.000,B 0.000,C 90.000,E1 112.333} C_DIS
LIN {X -0.185,Y -672.436,Z 905.421,A 0.000,B 0.000,C 90.000,E1 111.844} C_DIS
LIN {X -0.064,Y -670.539,Z 905.421,A 0.000,B 0.000,C 90.000,E1 111.716} C_DIS
LIN {X -0.128,Y -668.995,Z 905.420,A 0.000,B 0.000,C 90.000,E1 111.663} C_DIS
LIN {X 0.067,Y -665.475,Z 905.420,A 0.000,B 0.000,C 90.000,E1 111.535} C_DIS
LIN {X 0.163,Y -662.456,Z 905.419,A 0.000,B 0.000,C 90.000,E1 111.408} C_DIS
LIN {X 0.005,Y -659.577,Z 905.419,A 0.000,B 0.000,C 90.000,E1 111.354} C_DIS
LIN {X 0.380,Y -656.514,Z 905.418,A 0.000,B 0.000,C 90.000,E1 111.280} C_DIS
LIN {X -0.095,Y -654.360,Z 905.418,A 0.000,B 0.000,C 90.000,E1 111.280} C_DIS
LIN {X 0.067,Y -644.420,Z 905.418,A 0.000,B 0.000,C 90.000,E1 111.153} C_DIS
LIN {X -0.126,Y -634.286,Z 905.417,A 0.000,B 0.000,C 90.000,E1 111.046} C_DIS
LIN {X 0.132,Y -628.517,Z 905.416,A 0.000,B 0.000,C 90.000,E1 110.918} C_DIS
LIN {X 0.017,Y -622.408,Z 905.416,A 0.000,B 0.000,C 90.000,E1 110.791} C_DIS
LIN {X -0.329,Y -619.055,Z 905.415,A 0.000,B 0.000,C 90.000,E1 110.737} C_DIS
LIN {X -0.085,Y -613.456,Z 905.414,A 0.000,B 0.000,C 90.000,E1 110.536} C_DIS
LIN {X -0.048,Y -606.279,Z 905.413,A 0.000,B 0.000,C 90.000,E1 110.248} C_DIS
LIN {X 0.257,Y -600.500,Z 905.411,A 0.000,B 0.000,C 90.000,E1 109.939} C_DIS
LIN {X 0.192,Y -585.063,Z 905.406,A 0.000,B 0.000,C 90.000,E1 109.033} C_DIS
LIN {X -0.074,Y -580.237,Z 905.404,A 0.000,B 0.000,C 90.000,E1 108.779} C_DIS
LIN {X 0.103,Y -573.211,Z 905.402,A 0.000,B 0.000,C 90.000,E1 108.417} C_DIS
LIN {X 0.166,Y -567.490,Z 905.401,A 0.000,B 0.000,C 90.000,E1 108.181} C_DIS
LIN {X 0.007,Y -562.232,Z 905.400,A 0.000,B 0.000,C 90.000,E1 108.000} C_DIS
LIN {X -0.072,Y -556.842,Z 905.399,A 0.000,B 0.000,C 90.000,E1 107.764} C_DIS
LIN {X -0.112,Y -556.770,Z 905.399,A 0.000,B 0.000,C 90.000,E1 107.764} C_DIS
LIN {X -0.096,Y -555.352,Z 905.398,A 0.000,B 0.000,C 90.000,E1 107.583} C_DIS
LIN {X -0.138,Y -555.339,Z 905.398,A 0.000,B 0.000,C 90.000,E1 107.583} C_DIS
LIN {X 0.164,Y -554.913,Z 905.396,A 0.000,B 0.000,C 90.000,E1 107.330} C_DIS
LIN {X -0.252,Y -554.745,Z 905.395,A 0.000,B 0.000,C 90.000,E1 107.094} C_DIS
LIN {X 0.139,Y -554.764,Z 905.392,A 0.000,B 0.000,C 90.000,E1 106.496} C_DIS
LIN {X 0.093,Y -555.352,Z 905.383,A 0.000,B 0.000,C 90.000,E1 104.828} C_DIS
LIN {X 0.047,Y -556.340,Z 905.372,A 0.000,B 0.000,C 90.000,E1 102.883} C_DIS
LIN {X -0.095,Y -557.597,Z 905.361,A 0.000,B 0.000,C 90.000,E1 100.950} C_DIS
LIN {X 0.096,Y -558.815,Z 905.352,A 0.000,B 0.000,C 90.000,E1 99.265} C_DIS
LIN {X 0.165,Y -559.797,Z 905.344,A 0.000,B 0.000,C 90.000,E1 97.871} C_DIS
LIN {X 0.170,Y -560.672,Z 905.336,A 0.000,B 0.000,C 90.000,E1 96.486} C_DIS
LIN {X 0.220,Y -561.624,Z 905.327,A 0.000,B 0.000,C 90.000,E1 94.821} C_DIS
LIN {X 0.207,Y -562.289,Z 905.319,A 0.000,B 0.000,C 90.000,E1 93.440} C_DIS
LIN {X 0.171,Y -562.886,Z 905.312,A 0.000,B 0.000,C 90.000,E1 92.064} C_DIS
LIN {X 0.245,Y -563.374,Z 905.302,A 0.000,B 0.000,C 90.000,E1 90.401} C_DIS
LIN {X 0.105,Y -563.703,Z 905.296,A 0.000,B 0.000,C 90.000,E1 89.312} C_DIS
LIN {X 0.195,Y -564.046,Z 905.287,A 0.000,B 0.000,C 90.000,E1 87.650} C_DIS
LIN {X -0.136,Y -564.363,Z 905.276,A 0.000,B 0.000,C 90.000,E1 85.755} C_DIS
LIN {X -0.008,Y -564.639,Z 905.267,A 0.000,B 0.000,C 90.000,E1 84.090} C_DIS
LIN {X -0.075,Y -564.840,Z 905.261,A 0.000,B 0.000,C 90.000,E1 82.996} C_DIS
LIN {X -0.050,Y -565.474,Z 905.249,A 0.000,B 0.000,C 90.000,E1 80.792} C_DIS
LIN {X 0.272,Y -566.457,Z 905.235,A 0.000,B 0.000,C 90.000,E1 78.285} C_DIS
LIN {X 0.033,Y -567.171,Z 905.227,A 0.000,B 0.000,C 90.000,E1 76.937} C_DIS
LIN {X 0.114,Y -568.049,Z 905.218,A 0.000,B 0.000,C 90.000,E1 75.283} C_DIS
LIN {X 0.033,Y -568.680,Z 905.211,A 0.000,B 0.000,C 90.000,E1 73.921} C_DIS
LIN {X 0.115,Y -569.260,Z 905.203,A 0.000,B 0.000,C 90.000,E1 72.543} C_DIS
LIN {X -0.336,Y -569.729,Z 905.196,A 0.000,B 0.000,C 90.000,E1 71.221} C_DIS
LIN {X -0.062,Y -570.069,Z 905.188,A 0.000,B 0.000,C 90.000,E1 69.826} C_DIS
LIN {X 0.238,Y -570.427,Z 905.179,A 0.000,B 0.000,C 90.000,E1 68.156} C_DIS
LIN {X 0.027,Y -570.654,Z 905.170,A 0.000,B 0.000,C 90.000,E1 66.538} C_DIS
LIN {X -0.019,Y -570.693,Z 905.162,A 0.000,B 0.000,C 90.000,E1 65.177} C_DIS
LIN {X -0.101,Y -570.760,Z 905.155,A 0.000,B 0.000,C 90.000,E1 63.819} C_DIS
LIN {X 0.077,Y -570.709,Z 905.147,A 0.000,B 0.000,C 90.000,E1 62.436} C_DIS
LIN {X -0.334,Y -570.639,Z 905.141,A 0.000,B 0.000,C 90.000,E1 61.385} C_DIS
LIN {X -0.311,Y -570.420,Z 905.132,A 0.000,B 0.000,C 90.000,E1 59.744} C_DIS
LIN {X 0.173,Y -570.028,Z 905.124,A 0.000,B 0.000,C 90.000,E1 58.329} C_DIS
LIN {X 0.049,Y -569.475,Z 905.118,A 0.000,B 0.000,C 90.000,E1 57.248} C_DIS
LIN {X 0.034,Y -568.693,Z 905.111,A 0.000,B 0.000,C 90.000,E1 55.881} C_DIS
LIN {X 0.079,Y -568.072,Z 905.106,A 0.000,B 0.000,C 90.000,E1 55.055} C_DIS
LIN {X -0.140,Y -567.655,Z 905.103,A 0.000,B 0.000,C 90.000,E1 54.529} C_DIS
LIN {X 0.012,Y -566.499,Z 905.097,A 0.000,B 0.000,C 90.000,E1 53.417} C_DIS
LIN {X 0.030,Y -565.164,Z 905.091,A 0.000,B 0.000,C 90.000,E1 52.316} C_DIS
LIN {X -0.318,Y -563.605,Z 905.085,A 0.000,B 0.000,C 90.000,E1 51.251} C_DIS
LIN {X 0.349,Y -562.258,Z 905.080,A 0.000,B 0.000,C 90.000,E1 50.356} C_DIS
LIN {X 0.210,Y -560.701,Z 905.075,A 0.000,B 0.000,C 90.000,E1 49.542} C_DIS
LIN {X -0.036,Y -559.578,Z 905.072,A 0.000,B 0.000,C 90.000,E1 49.013} C_DIS
LIN {X 0.161,Y -557.619,Z 905.068,A 0.000,B 0.000,C 90.000,E1 48.162} C_DIS
LIN {X 0.338,Y -555.346,Z 905.063,A 0.000,B 0.000,C 90.000,E1 47.310} C_DIS
LIN {X 0.086,Y -552.782,Z 905.058,A 0.000,B 0.000,C 90.000,E1 46.500} C_DIS
LIN {X -0.215,Y -550.951,Z 905.055,A 0.000,B 0.000,C 90.000,E1 45.972} C_DIS
LIN {X 0.269,Y -547.890,Z 905.051,A 0.000,B 0.000,C 90.000,E1 45.081} C_DIS
LIN {X 0.314,Y -545.708,Z 905.048,A 0.000,B 0.000,C 90.000,E1 44.514} C_DIS
LIN {X -0.230,Y -542.670,Z 905.044,A 0.000,B 0.000,C 90.000,E1 43.866} C_DIS
LIN {X -0.038,Y -539.228,Z 905.040,A 0.000,B 0.000,C 90.000,E1 43.137} C_DIS
LIN {X 0.330,Y -536.330,Z 905.036,A 0.000,B 0.000,C 90.000,E1 42.528} C_DIS
LIN {X -0.078,Y -533.234,Z 905.033,A 0.000,B 0.000,C 90.000,E1 42.000} C_DIS
LIN {X 0.014,Y -529.032,Z 905.029,A 0.000,B 0.000,C 90.000,E1 41.272} C_DIS
LIN {X 0.147,Y -526.424,Z 905.027,A 0.000,B 0.000,C 90.000,E1 40.825} C_DIS
LIN {X 0.175,Y -519.780,Z 905.021,A 0.000,B 0.000,C 90.000,E1 39.806} C_DIS
LIN {X -0.008,Y -515.732,Z 905.018,A 0.000,B 0.000,C 90.000,E1 39.241} C_DIS
LIN {X -0.148,Y -511.461,Z 905.015,A 0.000,B 0.000,C 90.000,E1 38.669} C_DIS
LIN {X 0.196,Y -505.647,Z 905.011,A 0.000,B 0.000,C 90.000,E1 37.890} C_DIS
LIN {X -0.010,Y -500.655,Z 905.007,A 0.000,B 0.000,C 90.000,E1 37.317} C_DIS
LIN {X -0.123,Y -494.154,Z 905.003,A 0.000,B 0.000,C 90.000,E1 36.583} C_DIS
LIN {X -0.172,Y -488.673,Z 905.000,A 0.000,B 0.000,C 90.000,E1 36.011} C_DIS
LIN {X 0.063,Y -483.180,Z 904.997,A 0.000,B 0.000,C 90.000,E1 35.438} C_DIS
LIN {X 0.182,Y -475.828,Z 904.993,A 0.000,B 0.000,C 90.000,E1 34.739} C_DIS
LIN {X -0.201,Y -466.902,Z 904.989,A 0.000,B 0.000,C 90.000,E1 33.992} C_DIS
LIN {X 0.236,Y -457.809,Z 904.984,A 0.000,B 0.000,C 90.000,E1 33.166} C_DIS
LIN {X 0.050,Y -448.525,Z 904.980,A 0.000,B 0.000,C 90.000,E1 32.418} C_DIS
LIN {X 0.175,Y -434.588,Z 904.974,A 0.000,B 0.000,C 90.000,E1 31.258} C_DIS
LIN {X 0.107,Y -419.323,Z 904.967,A 0.000,B 0.000,C 90.000,E1 29.951} C_DIS
LIN {X -0.174,Y -405.982,Z 904.960,A 0.000,B 0.000,C 90.000,E1 28.743} C_DIS
LIN {X 0.152,Y -400.138,Z 904.956,A 0.000,B 0.000,C 90.000,E1 28.103} C_DIS
LIN {X -0.057,Y -396.529,Z 904.954,A 0.000,B 0.000,C 90.000,E1 27.719} C_DIS
LIN {X 0.001,Y -393.123,Z 904.951,A 0.000,B 0.000,C 90.000,E1 27.257} C_DIS
LIN {X 0.098,Y -390.452,Z 904.948,A 0.000,B 0.000,C 90.000,E1 26.668} C_DIS
LIN {X -0.086,Y -389.221,Z 904.945,A 0.000,B 0.000,C 90.000,E1 26.027} C_DIS
LIN {X 0.120,Y -388.835,Z 904.941,A 0.000,B 0.000,C 90.000,E1 25.283} C_DIS
LIN {X 0.147,Y -389.063,Z 904.936,A 0.000,B 0.000,C 90.000,E1 24.387} C_DIS
LIN {X 0.153,Y -393.185,Z 904.910,A 0.000,B 0.000,C 90.000,E1 19.758} C_DIS
LIN {X -0.177,Y -396.916,Z 904.892,A 0.000,B 0.000,C 90.000,E1 16.622} C_DIS
LIN {X 0.083,Y -400.517,Z 904.877,A 0.000,B 0.000,C 90.000,E1 13.772} C_DIS
LIN {X -0.126,Y -405.028,Z 904.859,A 0.000,B 0.000,C 90.000,E1 10.658} C_DIS
LIN {X -0.032,Y -409.513,Z 904.844,A 0.000,B 0.000,C 90.000,E1 7.871} C_DIS
LIN {X 0.026,Y -413.193,Z 904.832,A 0.000,B 0.000,C 90.000,E1 5.796} C_DIS
LIN {X 0.196,Y -418.569,Z 904.817,A 0.000,B 0.000,C 90.000,E1 3.037} C_DIS
LIN {X 0.161,Y -425.878,Z 904.799,A 0.000,B 0.000,C 90.000,E1 359.771} C_DIS
LIN {X -0.161,Y -432.777,Z 904.784,A 0.000,B 0.000,C 90.000,E1 357.135} C_DIS
LIN {X -0.018,Y -434.479,Z 904.781,A 0.000,B 0.000,C 90.000,E1 356.617} C_DIS
LIN {X 0.067,Y -435.791,Z 904.779,A 0.000,B 0.000,C 90.000,E1 356.274} C_DIS
LIN {X 0.112,Y -436.598,Z 904.779,A 0.000,B 0.000,C 90.000,E1 356.102} C_DIS
LIN {X 0.002,Y -437.741,Z 904.777,A 0.000,B 0.000,C 90.000,E1 355.927} C_DIS
LIN {X 0.152,Y -441.854,Z 904.775,A 0.000,B 0.000,C 90.000,E1 355.412} C_DIS
LIN {X -0.043,Y -442.724,Z 904.774,A 0.000,B 0.000,C 90.000,E1 355.355} C_DIS
LIN {X -0.110,Y -447.206,Z 904.773,A 0.000,B 0.000,C 90.000,E1 355.065} C_DIS
LIN {X -0.050,Y -449.100,Z 904.772,A 0.000,B 0.000,C 90.000,E1 354.951} C_DIS
LIN {X -0.050,Y -461.823,Z 904.769,A 0.000,B 0.000,C 90.000,E1 354.375} C_DIS
LIN {X -0.202,Y -471.984,Z 904.766,A 0.000,B 0.000,C 90.000,E1 353.913} C_DIS
LIN {X 0.187,Y -483.561,Z 904.763,A 0.000,B 0.000,C 90.000,E1 353.280} C_DIS
LIN {X -0.110,Y -496.728,Z 904.759,A 0.000,B 0.000,C 90.000,E1 352.591} C_DIS
LIN {X -0.100,Y -504.921,Z 904.756,A 0.000,B 0.000,C 90.000,E1 352.129} C_DIS
LIN {X -0.115,Y -514.379,Z 904.753,A 0.000,B 0.000,C 90.000,E1 351.546} C_DIS
LIN {X -0.033,Y -522.196,Z 904.750,A 0.000,B 0.000,C 90.000,E1 351.027} C_DIS
LIN {X -0.003,Y -529.689,Z 904.747,A 0.000,B 0.000,C 90.000,E1 350.500} C_DIS
LIN {X 0.073,Y -537.007,Z 904.744,A 0.000,B 0.000,C 90.000,E1 349.926} C_DIS
LIN {X -0.092,Y -545.394,Z 904.740,A 0.000,B 0.000,C 90.000,E1 349.218} C_DIS
LIN {X -0.041,Y -552.063,Z 904.737,A 0.000,B 0.000,C 90.000,E1 348.578} C_DIS
LIN {X -0.054,Y -557.214,Z 904.734,A 0.000,B 0.000,C 90.000,E1 348.049} C_DIS
LIN {X -0.193,Y -562.144,Z 904.731,A 0.000,B 0.000,C 90.000,E1 347.521} C_DIS
LIN {X -0.135,Y -567.981,Z 904.727,A 0.000,B 0.000,C 90.000,E1 346.825} C_DIS
LIN {X -0.201,Y -572.469,Z 904.724,A 0.000,B 0.000,C 90.000,E1 346.284} C_DIS
LIN {X 0.290,Y -579.538,Z 904.718,A 0.000,B 0.000,C 90.000,E1 345.283} C_DIS
LIN {X -0.257,Y -586.015,Z 904.713,A 0.000,B 0.000,C 90.000,E1 344.393} C_DIS
LIN {X 0.143,Y -590.272,Z 904.709,A 0.000,B 0.000,C 90.000,E1 343.685} C_DIS
LIN {X -0.183,Y -596.541,Z 904.704,A 0.000,B 0.000,C 90.000,E1 342.653} C_DIS
LIN {X -0.034,Y -602.341,Z 904.698,A 0.000,B 0.000,C 90.000,E1 341.583} C_DIS
LIN {X -0.194,Y -607.784,Z 904.692,A 0.000,B 0.000,C 90.000,E1 340.550} C_DIS
LIN {X -0.283,Y -612.945,Z 904.686,A 0.000,B 0.000,C 90.000,E1 339.518} C_DIS
LIN {X -0.084,Y -617.807,Z 904.680,A 0.000,B 0.000,C 90.000,E1 338.465} C_DIS
LIN {X 0.184,Y -622.391,Z 904.675,A 0.000,B 0.000,C 90.000,E1 337.411} C_DIS
LIN {X -0.305,Y -627.629,Z 904.668,A 0.000,B 0.000,C 90.000,E1 336.177} C_DIS
LIN {X -0.274,Y -629.589,Z 904.665,A 0.000,B 0.000,C 90.000,E1 335.665} C_DIS
LIN {X 0.139,Y -633.312,Z 904.659,A 0.000,B 0.000,C 90.000,E1 334.613} C_DIS
LIN {X -0.273,Y -636.922,Z 904.653,A 0.000,B 0.000,C 90.000,E1 333.640} C_DIS
LIN {X -0.063,Y -640.211,Z 904.648,A 0.000,B 0.000,C 90.000,E1 332.615} C_DIS
LIN {X 0.188,Y -643.211,Z 904.642,A 0.000,B 0.000,C 90.000,E1 331.591} C_DIS
LIN {X -0.185,Y -647.354,Z 904.634,A 0.000,B 0.000,C 90.000,E1 330.127} C_DIS
LIN {X 0.000,Y -650.597,Z 904.627,A 0.000,B 0.000,C 90.000,E1 328.869} C_DIS
LIN {X 0.139,Y -653.011,Z 904.622,A 0.000,B 0.000,C 90.000,E1 327.867} C_DIS
LIN {X -0.246,Y -655.130,Z 904.616,A 0.000,B 0.000,C 90.000,E1 326.914} C_DIS
LIN {X 0.303,Y -656.927,Z 904.611,A 0.000,B 0.000,C 90.000,E1 325.881} C_DIS
LIN {X 0.337,Y -658.512,Z 904.605,A 0.000,B 0.000,C 90.000,E1 324.895} C_DIS
LIN {X 0.394,Y -659.837,Z 904.600,A 0.000,B 0.000,C 90.000,E1 323.909} C_DIS
LIN {X -0.016,Y -660.780,Z 904.596,A 0.000,B 0.000,C 90.000,E1 323.210} C_DIS
LIN {X -0.060,Y -661.794,Z 904.590,A 0.000,B 0.000,C 90.000,E1 322.236} C_DIS
LIN {X 0.028,Y -662.750,Z 904.585,A 0.000,B 0.000,C 90.000,E1 321.251} C_DIS
LIN {X 0.044,Y -664.360,Z 904.575,A 0.000,B 0.000,C 90.000,E1 319.542} C_DIS
LIN {X 0.045,Y -665.503,Z 904.569,A 0.000,B 0.000,C 90.000,E1 318.324} C_DIS
LIN {X -0.426,Y -666.539,Z 904.563,A 0.000,B 0.000,C 90.000,E1 317.391} C_DIS
LIN {X 0.057,Y -667.328,Z 904.559,A 0.000,B 0.000,C 90.000,E1 316.620} C_DIS
LIN {X 0.069,Y -668.242,Z 904.554,A 0.000,B 0.000,C 90.000,E1 315.648} C_DIS
LIN {X 0.114,Y -669.589,Z 904.546,A 0.000,B 0.000,C 90.000,E1 314.190} C_DIS
LIN {X -0.271,Y -671.116,Z 904.536,A 0.000,B 0.000,C 90.000,E1 312.528} C_DIS
LIN {X -0.158,Y -672.259,Z 904.529,A 0.000,B 0.000,C 90.000,E1 311.310} C_DIS
LIN {X -0.026,Y -673.220,Z 904.523,A 0.000,B 0.000,C 90.000,E1 310.092} C_DIS
LIN {X 0.222,Y -674.359,Z 904.515,A 0.000,B 0.000,C 90.000,E1 308.624} C_DIS
LIN {X -0.047,Y -675.335,Z 904.508,A 0.000,B 0.000,C 90.000,E1 307.443} C_DIS
LIN {X 0.226,Y -676.111,Z 904.501,A 0.000,B 0.000,C 90.000,E1 306.217} C_DIS
LIN {X -0.287,Y -676.883,Z 904.493,A 0.000,B 0.000,C 90.000,E1 304.818} C_DIS
LIN {X 0.100,Y -678.019,Z 904.481,A 0.000,B 0.000,C 90.000,E1 302.625} C_DIS
LIN {X 0.362,Y -679.190,Z 904.472,A 0.000,B 0.000,C 90.000,E1 300.924} C_DIS
LIN {X 0.166,Y -681.647,Z 904.457,A 0.000,B 0.000,C 90.000,E1 298.309} C_DIS
LIN {X -0.193,Y -683.698,Z 904.448,A 0.000,B 0.000,C 90.000,E1 296.668} C_DIS
LIN {X 0.180,Y -685.694,Z 904.440,A 0.000,B 0.000,C 90.000,E1 295.207} C_DIS
LIN {X 0.145,Y -686.892,Z 904.435,A 0.000,B 0.000,C 90.000,E1 294.259} C_DIS
LIN {X -0.099,Y -687.643,Z 904.431,A 0.000,B 0.000,C 90.000,E1 293.567} C_DIS
LIN {X 0.071,Y -687.834,Z 904.428,A 0.000,B 0.000,C 90.000,E1 293.078} C_DIS
LIN {X 0.293,Y -687.816,Z 904.427,A 0.000,B 0.000,C 90.000,E1 292.823} C_DIS
LIN {X -0.167,Y -687.034,Z 904.424,A 0.000,B 0.000,C 90.000,E1 292.386} C_DIS
LIN {X -0.209,Y -686.382,Z 904.423,A 0.000,B 0.000,C 90.000,E1 292.153} C_DIS
LIN {X 0.007,Y -684.964,Z 904.422,A 0.000,B 0.000,C 90.000,E1 291.897} C_DIS
LIN {X 0.065,Y -682.561,Z 904.420,A 0.000,B 0.000,C 90.000,E1 291.535} C_DIS
LIN {X 0.166,Y -681.437,Z 904.419,A 0.000,B 0.000,C 90.000,E1 291.408} C_DIS
LIN {X 0.264,Y -679.715,Z 904.418,A 0.000,B 0.000,C 90.000,E1 291.280} C_DIS
LIN {X 0.041,Y -671.780,Z 904.416,A 0.000,B 0.000,C 90.000,E1 290.918} C_DIS
LIN {X 0.290,Y -664.626,Z 904.415,A 0.000,B 0.000,C 90.000,E1 290.610} C_DIS
LIN {X -0.145,Y -660.375,Z 904.413,A 0.000,B 0.000,C 90.000,E1 290.429} C_DIS
LIN {X -0.205,Y -660.339,Z 904.413,A 0.000,B 0.000,C 90.000,E1 290.429} C_DIS
LIN {X -0.091,Y -659.974,Z 904.413,A 0.000,B 0.000,C 90.000,E1 290.355} C_DIS
LIN {X -0.135,Y -659.963,Z 904.413,A 0.000,B 0.000,C 90.000,E1 290.355} C_DIS
LIN {X 0.235,Y -660.006,Z 904.412,A 0.000,B 0.000,C 90.000,E1 290.120} C_DIS
LIN {X 0.290,Y -660.176,Z 904.411,A 0.000,B 0.000,C 90.000,E1 289.993} C_DIS
LIN {X 0.232,Y -661.280,Z 904.409,A 0.000,B 0.000,C 90.000,E1 289.631} C_DIS
LIN {X 0.133,Y -664.577,Z 904.405,A 0.000,B 0.000,C 90.000,E1 288.906} C_DIS
LIN {X 0.115,Y -670.920,Z 904.398,A 0.000,B 0.000,C 90.000,E1 287.692} C_DIS
LIN {X -0.093,Y -674.226,Z 904.394,A 0.000,B 0.000,C 90.000,E1 286.985} C_DIS
LIN {X -0.017,Y -676.159,Z 904.392,A 0.000,B 0.000,C 90.000,E1 286.496} C_DIS
LIN {X -0.171,Y -678.567,Z 904.388,A 0.000,B 0.000,C 90.000,E1 285.788} C_DIS
LIN {X -0.117,Y -680.469,Z 904.384,A 0.000,B 0.000,C 90.000,E1 285.064} C_DIS
LIN {X -0.259,Y -682.532,Z 904.378,A 0.000,B 0.000,C 90.000,E1 284.120} C_DIS
LIN {X 0.317,Y -683.783,Z 904.374,A 0.000,B 0.000,C 90.000,E1 283.355} C_DIS
LIN {X 0.216,Y -685.035,Z 904.369,A 0.000,B 0.000,C 90.000,E1 282.411} C_DIS
LIN {X 0.004,Y -685.682,Z 904.365,A 0.000,B 0.000,C 90.000,E1 281.715} C_DIS
LIN {X -0.038,Y -685.869,Z 904.362,A 0.000,B 0.000,C 90.000,E1 281.243} C_DIS
LIN {X -0.213,Y -685.830,Z 904.360,A 0.000,B 0.000,C 90.000,E1 280.782} C_DIS
LIN {X -0.260,Y -685.436,Z 904.357,A 0.000,B 0.000,C 90.000,E1 280.310} C_DIS
LIN {X -0.286,Y -685.134,Z 904.356,A 0.000,B 0.000,C 90.000,E1 280.074} C_DIS
LIN {X 0.216,Y -684.287,Z 904.353,A 0.000,B 0.000,C 90.000,E1 279.557} C_DIS
LIN {X 0.043,Y -683.073,Z 904.351,A 0.000,B 0.000,C 90.000,E1 279.095} C_DIS
LIN {X -0.031,Y -681.477,Z 904.348,A 0.000,B 0.000,C 90.000,E1 278.624} C_DIS
LIN {X -0.219,Y -679.556,Z 904.345,A 0.000,B 0.000,C 90.000,E1 278.163} C_DIS
LIN {X -0.364,Y -678.563,Z 904.344,A 0.000,B 0.000,C 90.000,E1 277.936} C_DIS
LIN {X 0.044,Y -675.051,Z 904.340,A 0.000,B 0.000,C 90.000,E1 277.182} C_DIS
LIN {X -0.180,Y -672.487,Z 904.337,A 0.000,B 0.000,C 90.000,E1 276.720} C_DIS
LIN {X 0.244,Y -669.672,Z 904.335,A 0.000,B 0.000,C 90.000,E1 276.201} C_DIS
LIN {X -0.019,Y -666.613,Z 904.332,A 0.000,B 0.000,C 90.000,E1 275.739} C_DIS
LIN {X -0.300,Y -663.186,Z 904.329,A 0.000,B 0.000,C 90.000,E1 275.277} C_DIS
LIN {X -0.041,Y -658.356,Z 904.326,A 0.000,B 0.000,C 90.000,E1 274.645} C_DIS
LIN {X 0.228,Y -654.008,Z 904.323,A 0.000,B 0.000,C 90.000,E1 274.131} C_DIS
LIN {X -0.136,Y -649.324,Z 904.320,A 0.000,B 0.000,C 90.000,E1 273.669} C_DIS
LIN {X 0.255,Y -644.226,Z 904.318,A 0.000,B 0.000,C 90.000,E1 273.154} C_DIS
LIN {X 0.291,Y -637.539,Z 904.315,A 0.000,B 0.000,C 90.000,E1 272.579} C_DIS
LIN {X -0.069,Y -630.313,Z 904.311,A 0.000,B 0.000,C 90.000,E1 272.064} C_DIS
LIN {X -0.122,Y -624.324,Z 904.309,A 0.000,B 0.000,C 90.000,E1 271.661} C_DIS
LIN {X 0.061,Y -618.089,Z 904.307,A 0.000,B 0.000,C 90.000,E1 271.260} C_DIS
LIN {X -0.295,Y -609.899,Z 904.305,A 0.000,B 0.000,C 90.000,E1 270.859} C_DIS
LIN {X -0.155,Y -603.097,Z 904.303,A 0.000,B 0.000,C 90.000,E1 270.516} C_DIS
LIN {X -0.214,Y -596.488,Z 904.301,A 0.000,B 0.000,C 90.000,E1 270.229} C_DIS
LIN {X -0.046,Y -591.009,Z 904.300,A 0.000,B 0.000,C 90.000,E1 270.000} C_DIS
LIN {X -0.195,Y -583.606,Z 904.299,A 0.000,B 0.000,C 90.000,E1 269.771} C_DIS
LIN {X -0.019,Y -578.171,Z 904.298,A 0.000,B 0.000,C 90.000,E1 269.599} C_DIS
LIN {X -0.257,Y -572.006,Z 904.297,A 0.000,B 0.000,C 90.000,E1 269.484} C_DIS
LIN {X -0.171,Y -565.443,Z 904.296,A 0.000,B 0.000,C 90.000,E1 269.370} C_DIS
LIN {X 0.206,Y -557.193,Z 904.296,A 0.000,B 0.000,C 90.000,E1 269.255} C_DIS
LIN {X -0.146,Y -552.436,Z 904.296,A 0.000,B 0.000,C 90.000,E1 269.255} C_DIS
LIN {X 0.178,Y -549.936,Z 904.295,A 0.000,B 0.000,C 90.000,E1 269.141} C_DIS
LIN {X 0.240,Y -545.450,Z 904.293,A 0.000,B 0.000,C 90.000,E1 268.682} C_DIS
LIN {X 0.200,Y -545.433,Z 904.293,A 0.000,B 0.000,C 90.000,E1 268.682} C_DIS
LIN {X -0.138,Y -544.192,Z 904.291,A 0.000,B 0.000,C 90.000,E1 268.339} C_DIS
LIN {X 0.054,Y -543.216,Z 904.287,A 0.000,B 0.000,C 90.000,E1 267.593} C_DIS
LIN {X -0.024,Y -540.212,Z 904.266,A 0.000,B 0.000,C 90.000,E1 263.913} C_DIS
LIN {X 0.046,Y -539.578,Z 904.261,A 0.000,B 0.000,C 90.000,E1 263.053} C_DIS
LIN {X -0.235,Y -538.335,Z 904.254,A 0.000,B 0.000,C 90.000,E1 261.659} C_DIS
LIN {X 0.005,Y -536.976,Z 904.246,A 0.000,B 0.000,C 90.000,E1 260.208} C_DIS
LIN {X -0.258,Y -535.186,Z 904.236,A 0.000,B 0.000,C 90.000,E1 258.522} C_DIS
LIN {X 0.007,Y -533.583,Z 904.228,A 0.000,B 0.000,C 90.000,E1 257.061} C_DIS
LIN {X -0.161,Y -531.797,Z 904.220,A 0.000,B 0.000,C 90.000,E1 255.644} C_DIS
LIN {X 0.117,Y -530.273,Z 904.214,A 0.000,B 0.000,C 90.000,E1 254.464} C_DIS
LIN {X 0.005,Y -528.892,Z 904.207,A 0.000,B 0.000,C 90.000,E1 253.323} C_DIS
LIN {X 0.053,Y -527.160,Z 904.199,A 0.000,B 0.000,C 90.000,E1 251.873} C_DIS
LIN {X -0.264,Y -524.617,Z 904.188,A 0.000,B 0.000,C 90.000,E1 249.880} C_DIS
LIN {X 0.195,Y -521.826,Z 904.177,A 0.000,B 0.000,C 90.000,E1 247.794} C_DIS
LIN {X -0.003,Y -519.745,Z 904.169,A 0.000,B 0.000,C 90.000,E1 246.357} C_DIS
LIN {X 0.249,Y -516.704,Z 904.157,A 0.000,B 0.000,C 90.000,E1 244.280} C_DIS
LIN {X -0.069,Y -515.352,Z 904.152,A 0.000,B 0.000,C 90.000,E1 243.435} C_DIS
LIN {X 0.174,Y -513.416,Z 904.146,A 0.000,B 0.000,C 90.000,E1 242.231} C_DIS
LIN {X 0.154,Y -510.280,Z 904.136,A 0.000,B 0.000,C 90.000,E1 240.461} C_DIS
LIN {X -0.052,Y -506.622,Z 904.125,A 0.000,B 0.000,C 90.000,E1 238.408} C_DIS
LIN {X 0.093,Y -504.410,Z 904.118,A 0.000,B 0.000,C 90.000,E1 237.199} C_DIS
LIN {X 0.174,Y -502.673,Z 904.113,A 0.000,B 0.000,C 90.000,E1 236.294} C_DIS
LIN {X 0.239,Y -500.706,Z 904.108,A 0.000,B 0.000,C 90.000,E1 235.388} C_DIS
LIN {X 0.026,Y -495.159,Z 904.095,A 0.000,B 0.000,C 90.000,E1 233.004} C_DIS
LIN {X 0.000,Y -491.759,Z 904.086,A 0.000,B 0.000,C 90.000,E1 231.492} C_DIS
LIN {X -0.012,Y -487.737,Z 904.076,A 0.000,B 0.000,C 90.000,E1 229.666} C_DIS
LIN {X -0.060,Y -485.036,Z 904.069,A 0.000,B 0.000,C 90.000,E1 228.447} C_DIS
LIN {X 0.039,Y -479.503,Z 904.055,A 0.000,B 0.000,C 90.000,E1 225.972} C_DIS
LIN {X -0.045,Y -476.022,Z 904.047,A 0.000,B 0.000,C 90.000,E1 224.433} C_DIS
LIN {X 0.240,Y -471.714,Z 904.036,A 0.000,B 0.000,C 90.000,E1 222.528} C_DIS
LIN {X -0.210,Y -467.525,Z 904.026,A 0.000,B 0.000,C 90.000,E1 220.701} C_DIS
LIN {X -0.149,Y -464.095,Z 904.017,A 0.000,B 0.000,C 90.000,E1 219.116} C_DIS
LIN {X 0.164,Y -461.476,Z 904.010,A 0.000,B 0.000,C 90.000,E1 217.810} C_DIS
LIN {X -0.092,Y -457.455,Z 904.000,A 0.000,B 0.000,C 90.000,E1 215.931} C_DIS
LIN {X -0.063,Y -454.009,Z 903.991,A 0.000,B 0.000,C 90.000,E1 214.326} C_DIS
LIN {X -0.265,Y -449.724,Z 903.980,A 0.000,B 0.000,C 90.000,E1 212.418} C_DIS
LIN {X -0.182,Y -445.502,Z 903.969,A 0.000,B 0.000,C 90.000,E1 210.463} C_DIS
LIN {X -0.047,Y -441.306,Z 903.958,A 0.000,B 0.000,C 90.000,E1 208.487} C_DIS
LIN {X -0.006,Y -436.137,Z 903.945,A 0.000,B 0.000,C 90.000,E1 206.181} C_DIS
LIN {X 0.073,Y -432.575,Z 903.936,A 0.000,B 0.000,C 90.000,E1 204.515} C_DIS
LIN {X 0.093,Y -428.215,Z 903.925,A 0.000,B 0.000,C 90.000,E1 202.514} C_DIS
LIN {X 0.049,Y -424.701,Z 903.916,A 0.000,B 0.000,C 90.000,E1 200.844} C_DIS
LIN {X 0.180,Y -421.187,Z 903.907,A 0.000,B 0.000,C 90.000,E1 199.141} C_DIS
LIN {X 0.107,Y -417.763,Z 903.897,A 0.000,B 0.000,C 90.000,E1 197.457} C_DIS
LIN {X -0.003,Y -413.658,Z 903.886,A 0.000,B 0.000,C 90.000,E1 195.426} C_DIS
LIN {X 0.077,Y -409.499,Z 903.874,A 0.000,B 0.000,C 90.000,E1 193.355} C_DIS
LIN {X -0.135,Y -406.259,Z 903.865,A 0.000,B 0.000,C 90.000,E1 191.658} C_DIS
LIN {X -0.013,Y -402.825,Z 903.855,A 0.000,B 0.000,C 90.000,E1 189.905} C_DIS
LIN {X -0.052,Y -398.535,Z 903.843,A 0.000,B 0.000,C 90.000,E1 187.814} C_DIS
LIN {X -0.070,Y -392.612,Z 903.826,A 0.000,B 0.000,C 90.000,E1 184.645} C_DIS
LIN {X -0.002,Y -387.298,Z 903.808,A 0.000,B 0.000,C 90.000,E1 181.432} C_DIS
LIN {X -0.005,Y -384.989,Z 903.800,A 0.000,B 0.000,C 90.000,E1 180.000} C_DIS
LIN {X -0.158,Y -382.204,Z 903.790,A 0.000,B 0.000,C 90.000,E1 178.224} C_DIS
LIN {X -0.060,Y -377.563,Z 903.772,A 0.000,B 0.000,C 90.000,E1 174.951} C_DIS
LIN {X 0.077,Y -376.322,Z 903.762,A 0.000,B 0.000,C 90.000,E1 173.109} C_DIS
LIN {X -0.132,Y -376.481,Z 903.758,A 0.000,B 0.000,C 90.000,E1 172.527} C_DIS
LIN {X -0.007,Y -377.134,Z 903.754,A 0.000,B 0.000,C 90.000,E1 171.781} C_DIS
LIN {X -0.113,Y -377.580,Z 903.752,A 0.000,B 0.000,C 90.000,E1 171.432} C_DIS
LIN {X 0.156,Y -378.361,Z 903.750,A 0.000,B 0.000,C 90.000,E1 171.027} C_DIS
LIN {X 0.053,Y -379.324,Z 903.748,A 0.000,B 0.000,C 90.000,E1 170.679} C_DIS
LIN {X -0.016,Y -381.308,Z 903.745,A 0.000,B 0.000,C 90.000,E1 170.151} C_DIS
LIN {X -0.107,Y -383.030,Z 903.743,A 0.000,B 0.000,C 90.000,E1 169.803} C_DIS
LIN {X -0.186,Y -384.167,Z 903.742,A 0.000,B 0.000,C 90.000,E1 169.634} C_DIS
LIN {X -0.008,Y -388.406,Z 903.739,A 0.000,B 0.000,C 90.000,E1 169.050} C_DIS
LIN {X -0.065,Y -392.394,Z 903.737,A 0.000,B 0.000,C 90.000,E1 168.701} C_DIS
LIN {X 0.116,Y -395.783,Z 903.736,A 0.000,B 0.000,C 90.000,E1 168.409} C_DIS
LIN {X 0.008,Y -402.139,Z 903.733,A 0.000,B 0.000,C 90.000,E1 167.993} C_DIS
LIN {X 0.150,Y -410.264,Z 903.731,A 0.000,B 0.000,C 90.000,E1 167.465} C_DIS
LIN {X 0.092,Y -418.502,Z 903.728,A 0.000,B 0.000,C 90.000,E1 166.937} C_DIS
LIN {X -0.068,Y -424.977,Z 903.725,A 0.000,B 0.000,C 90.000,E1 166.520} C_DIS
LIN {X -0.125,Y -432.893,Z 903.722,A 0.000,B 0.000,C 90.000,E1 165.936} C_DIS
LIN {X 0.188,Y -439.110,Z 903.719,A 0.000,B 0.000,C 90.000,E1 165.408} C_DIS
LIN {X 0.194,Y -448.090,Z 903.715,A 0.000,B 0.000,C 90.000,E1 164.629} C_DIS
LIN {X 0.108,Y -455.453,Z 903.711,A 0.000,B 0.000,C 90.000,E1 163.976} C_DIS
LIN {X 0.157,Y -459.804,Z 903.709,A 0.000,B 0.000,C 90.000,E1 163.559} C_DIS
LIN {X -0.005,Y -465.437,Z 903.706,A 0.000,B 0.000,C 90.000,E1 163.015} C_DIS
LIN {X -0.114,Y -474.989,Z 903.700,A 0.000,B 0.000,C 90.000,E1 162.000} C_DIS
LIN {X -0.196,Y -481.574,Z 903.696,A 0.000,B 0.000,C 90.000,E1 161.275} C_DIS
LIN {X -0.235,Y -491.459,Z 903.689,A 0.000,B 0.000,C 90.000,E1 160.061} C_DIS
LIN {X 0.171,Y -499.346,Z 903.683,A 0.000,B 0.000,C 90.000,E1 158.954} C_DIS
LIN {X -0.070,Y -504.968,Z 903.679,A 0.000,B 0.000,C 90.000,E1 158.230} C_DIS
LIN {X 0.106,Y -509.099,Z 903.676,A 0.000,B 0.000,C 90.000,E1 157.614} C_DIS
LIN {X 0.235,Y -523.218,Z 903.664,A 0.000,B 0.000,C 90.000,E1 155.537} C_DIS
LIN {X -0.063,Y -530.768,Z 903.658,A 0.000,B 0.000,C 90.000,E1 154.409} C_DIS
LIN {X 0.039,Y -540.582,Z 903.649,A 0.000,B 0.000,C 90.000,E1 152.820} C_DIS
LIN {X -0.137,Y -547.803,Z 903.642,A 0.000,B 0.000,C 90.000,E1 151.563} C_DIS
LIN {X 0.069,Y -556.255,Z 903.633,A 0.000,B 0.000,C 90.000,E1 149.999} C_DIS
LIN {X -0.064,Y -566.146,Z 903.623,A 0.000,B 0.000,C 90.000,E1 148.074} C_DIS
LIN {X -0.134,Y -570.909,Z 903.617,A 0.000,B 0.000,C 90.000,E1 147.120} C_DIS
LIN {X 0.085,Y -576.007,Z 903.611,A 0.000,B 0.000,C 90.000,E1 146.008} C_DIS
LIN {X -0.177,Y -581.496,Z 903.604,A 0.000,B 0.000,C 90.000,E1 144.815} C_DIS
LIN {X 0.192,Y -586.275,Z 903.599,A 0.000,B 0.000,C 90.000,E1 143.703} C_DIS
LIN {X -0.250,Y -588.611,Z 903.596,A 0.000,B 0.000,C 90.000,E1 143.210} C_DIS
LIN {X -0.093,Y -596.349,Z 903.585,A 0.000,B 0.000,C 90.000,E1 141.331} C_DIS
LIN {X 0.167,Y -604.048,Z 903.575,A 0.000,B 0.000,C 90.000,E1 139.461} C_DIS
LIN {X -0.021,Y -612.872,Z 903.563,A 0.000,B 0.000,C 90.000,E1 137.391} C_DIS
LIN {X -0.091,Y -616.241,Z 903.559,A 0.000,B 0.000,C 90.000,E1 136.620} C_DIS
LIN {X -0.002,Y -621.891,Z 903.552,A 0.000,B 0.000,C 90.000,E1 135.324} C_DIS
LIN {X 0.059,Y -628.388,Z 903.543,A 0.000,B 0.000,C 90.000,E1 133.785} C_DIS
LIN {X -0.082,Y -633.743,Z 903.536,A 0.000,B 0.000,C 90.000,E1 132.528} C_DIS
LIN {X 0.339,Y -638.960,Z 903.529,A 0.000,B 0.000,C 90.000,E1 131.229} C_DIS
LIN {X -0.366,Y -642.086,Z 903.525,A 0.000,B 0.000,C 90.000,E1 130.539} C_DIS
LIN {X 0.122,Y -648.799,Z 903.515,A 0.000,B 0.000,C 90.000,E1 128.749} C_DIS
LIN {X -0.096,Y -654.490,Z 903.507,A 0.000,B 0.000,C 90.000,E1 127.282} C_DIS
LIN {X -0.032,Y -657.224,Z 903.503,A 0.000,B 0.000,C 90.000,E1 126.537} C_DIS
LIN {X 0.439,Y -662.466,Z 903.495,A 0.000,B 0.000,C 90.000,E1 125.025} C_DIS
LIN {X 0.175,Y -665.745,Z 903.489,A 0.000,B 0.000,C 90.000,E1 124.072} C_DIS
LIN {X 0.323,Y -668.851,Z 903.484,A 0.000,B 0.000,C 90.000,E1 123.086} C_DIS
LIN {X 0.141,Y -671.682,Z 903.479,A 0.000,B 0.000,C 90.000,E1 122.133} C_DIS
LIN {X -0.012,Y -674.025,Z 903.473,A 0.000,B 0.000,C 90.000,E1 121.180} C_DIS
LIN {X -0.307,Y -676.586,Z 903.467,A 0.000,B 0.000,C 90.000,E1 120.001} C_DIS
LIN {X 0.176,Y -678.228,Z 903.461,A 0.000,B 0.000,C 90.000,E1 118.999} C_DIS
LIN {X 0.031,Y -679.703,Z 903.456,A 0.000,B 0.000,C 90.000,E1 118.052} C_DIS
LIN {X -0.372,Y -680.853,Z 903.451,A 0.000,B 0.000,C 90.000,E1 117.129} C_DIS
LIN {X -0.168,Y -681.564,Z 903.445,A 0.000,B 0.000,C 90.000,E1 116.155} C_DIS
LIN {X -0.053,Y -681.931,Z 903.439,A 0.000,B 0.000,C 90.000,E1 114.951} C_DIS
LIN {X 0.278,Y -681.883,Z 903.435,A 0.000,B 0.000,C 90.000,E1 114.207} C_DIS
LIN {X -0.213,Y -681.663,Z 903.432,A 0.000,B 0.000,C 90.000,E1 113.770} C_DIS
LIN {X 0.192,Y -681.012,Z 903.429,A 0.000,B 0.000,C 90.000,E1 113.259} C_DIS
LIN {X 0.125,Y -680.421,Z 903.428,A 0.000,B 0.000,C 90.000,E1 113.025} C_DIS
LIN {X 0.322,Y -679.557,Z 903.427,A 0.000,B 0.000,C 90.000,E1 112.770} C_DIS
LIN {X -0.370,Y -678.559,Z 903.425,A 0.000,B 0.000,C 90.000,E1 112.589} C_DIS
LIN {X -0.274,Y -677.881,Z 903.425,A 0.000,B 0.000,C 90.000,E1 112.461} C_DIS
LIN {X -0.179,Y -676.847,Z 903.424,A 0.000,B 0.000,C 90.000,E1 112.333} C_DIS
LIN {X -0.086,Y -675.491,Z 903.423,A 0.000,B 0.000,C 90.000,E1 112.206} C_DIS
LIN {X 0.321,Y -672.959,Z 903.422,A 0.000,B 0.000,C 90.000,E1 111.897} C_DIS
LIN {X 0.155,Y -671.527,Z 903.421,A 0.000,B 0.000,C 90.000,E1 111.791} C_DIS
LIN {X 0.240,Y -669.151,Z 903.421,A 0.000,B 0.000,C 90.000,E1 111.663} C_DIS
LIN {X -0.060,Y -663.220,Z 903.419,A 0.000,B 0.000,C 90.000,E1 111.461} C_DIS
LIN {X -0.216,Y -660.935,Z 903.419,A 0.000,B 0.000,C 90.000,E1 111.408} C_DIS
LIN {X 0.291,Y -654.029,Z 903.418,A 0.000,B 0.000,C 90.000,E1 111.227} C_DIS
LIN {X -0.060,Y -636.853,Z 903.417,A 0.000,B 0.000,C 90.000,E1 111.046} C_DIS
LIN {X 0.256,Y -630.608,Z 903.416,A 0.000,B 0.000,C 90.000,E1 110.918} C_DIS
LIN {X 0.211,Y -624.317,Z 903.416,A 0.000,B 0.000,C 90.000,E1 110.791} C_DIS
LIN {X -0.119,Y -618.357,Z 903.415,A 0.000,B 0.000,C 90.000,E1 110.663} C_DIS
LIN {X -0.195,Y -612.554,Z 903.414,A 0.000,B 0.000,C 90.000,E1 110.482} C_DIS
LIN {X -0.143,Y -606.866,Z 903.412,A 0.000,B 0.000,C 90.000,E1 110.248} C_DIS
LIN {X -0.238,Y -601.246,Z 903.411,A 0.000,B 0.000,C 90.000,E1 109.993} C_DIS
LIN {X -0.170,Y -589.723,Z 903.407,A 0.000,B 0.000,C 90.000,E1 109.322} C_DIS
LIN {X -0.221,Y -580.211,Z 903.404,A 0.000,B 0.000,C 90.000,E1 108.779} C_DIS
LIN {X 0.012,Y -573.219,Z 903.402,A 0.000,B 0.000,C 90.000,E1 108.417} C_DIS
LIN {X 0.008,Y -565.672,Z 903.401,A 0.000,B 0.000,C 90.000,E1 108.127} C_DIS
LIN {X -0.019,Y -562.241,Z 903.400,A 0.000,B 0.000,C 90.000,E1 108.000} C_DIS
LIN {X -0.014,Y -557.112,Z 903.399,A 0.000,B 0.000,C 90.000,E1 107.764} C_DIS
LIN {X -0.060,Y -557.063,Z 903.399,A 0.000,B 0.000,C 90.000,E1 107.764} C_DIS
LIN {X -0.035,Y -555.649,Z 903.398,A 0.000,B 0.000,C 90.000,E1 107.583} C_DIS
LIN {X -0.077,Y -555.619,Z 903.398,A 0.000,B 0.000,C 90.000,E1 107.583} C_DIS
LIN {X 0.014,Y -555.153,Z 903.396,A 0.000,B 0.000,C 90.000,E1 107.330} C_DIS
LIN {X -0.240,Y -554.975,Z 903.395,A 0.000,B 0.000,C 90.000,E1 107.040} C_DIS
LIN {X 0.154,Y -554.997,Z 903.391,A 0.000,B 0.000,C 90.000,E1 106.441} C_DIS
LIN {X 0.244,Y -555.676,Z 903.381,A 0.000,B 0.000,C 90.000,E1 104.481} C_DIS
LIN {X 0.216,Y -556.723,Z 903.370,A 0.000,B 0.000,C 90.000,E1 102.535} C_DIS
LIN {X 0.228,Y -558.222,Z 903.357,A 0.000,B 0.000,C 90.000,E1 100.310} C_DIS
LIN {X -0.122,Y -559.454,Z 903.348,A 0.000,B 0.000,C 90.000,E1 98.681} C_DIS
LIN {X -0.123,Y -560.376,Z 903.341,A 0.000,B 0.000,C 90.000,E1 97.296} C_DIS
LIN {X -0.107,Y -561.180,Z 903.333,A 0.000,B 0.000,C 90.000,E1 95.910} C_DIS
LIN {X -0.224,Y -561.811,Z 903.327,A 0.000,B 0.000,C 90.000,E1 94.816} C_DIS
LIN {X -0.280,Y -562.469,Z 903.319,A 0.000,B 0.000,C 90.000,E1 93.440} C_DIS
LIN {X 0.249,Y -563.056,Z 903.311,A 0.000,B 0.000,C 90.000,E1 92.007} C_DIS
LIN {X -0.237,Y -563.528,Z 903.302,A 0.000,B 0.000,C 90.000,E1 90.401} C_DIS
LIN {X 0.188,Y -563.838,Z 903.296,A 0.000,B 0.000,C 90.000,E1 89.255} C_DIS
LIN {X 0.281,Y -564.187,Z 903.287,A 0.000,B 0.000,C 90.000,E1 87.593} C_DIS
LIN {X -0.047,Y -564.506,Z 903.276,A 0.000,B 0.000,C 90.000,E1 85.698} C_DIS
LIN {X 0.082,Y -564.783,Z 903.267,A 0.000,B 0.000,C 90.000,E1 84.033} C_DIS
LIN {X 0.084,Y -564.994,Z 903.261,A 0.000,B 0.000,C 90.000,E1 82.932} C_DIS
LIN {X 0.041,Y -565.631,Z 903.249,A 0.000,B 0.000,C 90.000,E1 80.735} C_DIS
LIN {X -0.190,Y -566.613,Z 903.235,A 0.000,B 0.000,C 90.000,E1 78.285} C_DIS
LIN {X 0.126,Y -567.314,Z 903.227,A 0.000,B 0.000,C 90.000,E1 76.881} C_DIS
LIN {X 0.207,Y -568.200,Z 903.218,A 0.000,B 0.000,C 90.000,E1 75.227} C_DIS
LIN {X 0.123,Y -568.809,Z 903.211,A 0.000,B 0.000,C 90.000,E1 73.866} C_DIS
LIN {X 0.000,Y -569.456,Z 903.201,A 0.000,B 0.000,C 90.000,E1 72.236} C_DIS
LIN {X -0.066,Y -569.809,Z 903.195,A 0.000,B 0.000,C 90.000,E1 71.148} C_DIS
LIN {X 0.218,Y -570.131,Z 903.188,A 0.000,B 0.000,C 90.000,E1 69.752} C_DIS
LIN {X -0.213,Y -570.477,Z 903.179,A 0.000,B 0.000,C 90.000,E1 68.156} C_DIS
LIN {X 0.100,Y -570.691,Z 903.169,A 0.000,B 0.000,C 90.000,E1 66.485} C_DIS
LIN {X 0.121,Y -570.729,Z 903.160,A 0.000,B 0.000,C 90.000,E1 64.845} C_DIS
LIN {X -0.038,Y -570.787,Z 903.154,A 0.000,B 0.000,C 90.000,E1 63.768} C_DIS
LIN {X 0.228,Y -570.700,Z 903.145,A 0.000,B 0.000,C 90.000,E1 62.103} C_DIS
LIN {X -0.180,Y -570.567,Z 903.139,A 0.000,B 0.000,C 90.000,E1 61.051} C_DIS
LIN {X 0.020,Y -570.359,Z 903.132,A 0.000,B 0.000,C 90.000,E1 59.665} C_DIS
LIN {X -0.277,Y -569.949,Z 903.124,A 0.000,B 0.000,C 90.000,E1 58.329} C_DIS
LIN {X 0.077,Y -569.361,Z 903.118,A 0.000,B 0.000,C 90.000,E1 57.199} C_DIS
LIN {X 0.372,Y -568.549,Z 903.110,A 0.000,B 0.000,C 90.000,E1 55.801} C_DIS
LIN {X -0.049,Y -567.921,Z 903.106,A 0.000,B 0.000,C 90.000,E1 55.022} C_DIS
LIN {X -0.132,Y -567.494,Z 903.103,A 0.000,B 0.000,C 90.000,E1 54.482} C_DIS
LIN {X 0.011,Y -566.293,Z 903.097,A 0.000,B 0.000,C 90.000,E1 53.371} C_DIS
LIN {X 0.020,Y -564.929,Z 903.090,A 0.000,B 0.000,C 90.000,E1 52.271} C_DIS
LIN {X -0.092,Y -563.801,Z 903.086,A 0.000,B 0.000,C 90.000,E1 51.457} C_DIS
LIN {X -0.111,Y -561.955,Z 903.080,A 0.000,B 0.000,C 90.000,E1 50.356} C_DIS
LIN {X 0.082,Y -560.986,Z 903.077,A 0.000,B 0.000,C 90.000,E1 49.784} C_DIS
LIN {X 0.289,Y -559.250,Z 903.072,A 0.000,B 0.000,C 90.000,E1 48.933} C_DIS
LIN {X 0.143,Y -556.435,Z 903.066,A 0.000,B 0.000,C 90.000,E1 47.838} C_DIS
LIN {X -0.130,Y -554.876,Z 903.063,A 0.000,B 0.000,C 90.000,E1 47.310} C_DIS
LIN {X 0.016,Y -552.243,Z 903.058,A 0.000,B 0.000,C 90.000,E1 46.458} C_DIS
LIN {X 0.092,Y -550.374,Z 903.055,A 0.000,B 0.000,C 90.000,E1 45.891} C_DIS
LIN {X -0.207,Y -547.268,Z 903.050,A 0.000,B 0.000,C 90.000,E1 45.081} C_DIS
LIN {X -0.165,Y -545.029,Z 903.047,A 0.000,B 0.000,C 90.000,E1 44.514} C_DIS
LIN {X 0.053,Y -541.893,Z 903.043,A 0.000,B 0.000,C 90.000,E1 43.785} C_DIS
LIN {X 0.049,Y -539.145,Z 903.040,A 0.000,B 0.000,C 90.000,E1 43.218} C_DIS
LIN {X -0.342,Y -536.230,Z 903.037,A 0.000,B 0.000,C 90.000,E1 42.690} C_DIS
LIN {X 0.181,Y -532.280,Z 903.033,A 0.000,B 0.000,C 90.000,E1 41.919} C_DIS
LIN {X 0.099,Y -528.914,Z 903.030,A 0.000,B 0.000,C 90.000,E1 41.353} C_DIS
LIN {X 0.043,Y -525.344,Z 903.027,A 0.000,B 0.000,C 90.000,E1 40.782} C_DIS
LIN {X -0.002,Y -518.614,Z 903.021,A 0.000,B 0.000,C 90.000,E1 39.769} C_DIS
LIN {X -0.123,Y -514.459,Z 903.018,A 0.000,B 0.000,C 90.000,E1 39.197} C_DIS
LIN {X 0.050,Y -510.048,Z 903.014,A 0.000,B 0.000,C 90.000,E1 38.588} C_DIS
LIN {X -0.128,Y -505.365,Z 903.011,A 0.000,B 0.000,C 90.000,E1 38.016} C_DIS
LIN {X 0.063,Y -500.383,Z 903.008,A 0.000,B 0.000,C 90.000,E1 37.397} C_DIS
LIN {X -0.023,Y -493.786,Z 903.004,A 0.000,B 0.000,C 90.000,E1 36.664} C_DIS
LIN {X 0.120,Y -487.179,Z 903.000,A 0.000,B 0.000,C 90.000,E1 35.964} C_DIS
LIN {X -0.031,Y -481.622,Z 902.997,A 0.000,B 0.000,C 90.000,E1 35.438} C_DIS
LIN {X 0.116,Y -474.262,Z 902.993,A 0.000,B 0.000,C 90.000,E1 34.739} C_DIS
LIN {X -0.227,Y -465.252,Z 902.989,A 0.000,B 0.000,C 90.000,E1 33.992} C_DIS
LIN {X -0.163,Y -453.044,Z 902.983,A 0.000,B 0.000,C 90.000,E1 32.959} C_DIS
LIN {X -0.013,Y -440.587,Z 902.977,A 0.000,B 0.000,C 90.000,E1 31.926} C_DIS
LIN {X -0.065,Y -423.675,Z 902.969,A 0.000,B 0.000,C 90.000,E1 30.512} C_DIS
LIN {X 0.206,Y -407.083,Z 902.961,A 0.000,B 0.000,C 90.000,E1 28.949} C_DIS
LIN {X -0.050,Y -401.351,Z 902.958,A 0.000,B 0.000,C 90.000,E1 28.409} C_DIS
LIN {X -0.089,Y -396.339,Z 902.955,A 0.000,B 0.000,C 90.000,E1 27.847} C_DIS
LIN {X 0.174,Y -394.044,Z 902.953,A 0.000,B 0.000,C 90.000,E1 27.513} C_DIS
LIN {X 0.124,Y -392.097,Z 902.951,A 0.000,B 0.000,C 90.000,E1 27.206} C_DIS
LIN {X 0.093,Y -390.147,Z 902.949,A 0.000,B 0.000,C 90.000,E1 26.744} C_DIS
LIN {X 0.030,Y -389.459,Z 902.946,A 0.000,B 0.000,C 90.000,E1 26.309} C_DIS
LIN {X -0.128,Y -389.075,Z 902.944,A 0.000,B 0.000,C 90.000,E1 25.976} C_DIS
LIN {X -0.173,Y -388.877,Z 902.940,A 0.000,B 0.000,C 90.000,E1 25.283} C_DIS
LIN {X -0.135,Y -389.294,Z 902.934,A 0.000,B 0.000,C 90.000,E1 24.207} C_DIS
LIN {X 0.157,Y -392.800,Z 902.913,A 0.000,B 0.000,C 90.000,E1 20.248} C_DIS
LIN {X -0.192,Y -395.553,Z 902.899,A 0.000,B 0.000,C 90.000,E1 17.819} C_DIS
LIN {X 0.022,Y -397.739,Z 902.889,A 0.000,B 0.000,C 90.000,E1 16.024} C_DIS
LIN {X -0.160,Y -400.925,Z 902.875,A 0.000,B 0.000,C 90.000,E1 13.592} C_DIS
LIN {X -0.046,Y -404.962,Z 902.860,A 0.000,B 0.000,C 90.000,E1 10.782} C_DIS
LIN {X 0.083,Y -410.005,Z 902.843,A 0.000,B 0.000,C 90.000,E1 7.644} C_DIS
LIN {X 0.196,Y -414.350,Z 902.829,A 0.000,B 0.000,C 90.000,E1 5.220} C_DIS
LIN {X -0.011,Y -420.540,Z 902.812,A 0.000,B 0.000,C 90.000,E1 2.178} C_DIS
LIN {X -0.209,Y -426.774,Z 902.797,A 0.000,B 0.000,C 90.000,E1 359.484} C_DIS
LIN {X -0.158,Y -432.840,Z 902.784,A 0.000,B 0.000,C 90.000,E1 357.135} C_DIS
LIN {X -0.014,Y -434.451,Z 902.781,A 0.000,B 0.000,C 90.000,E1 356.617} C_DIS
LIN {X 0.115,Y -436.426,Z 902.779,A 0.000,B 0.000,C 90.000,E1 356.102} C_DIS
LIN {X -0.198,Y -438.422,Z 902.777,A 0.000,B 0.000,C 90.000,E1 355.812} C_DIS
LIN {X 0.027,Y -439.865,Z 902.776,A 0.000,B 0.000,C 90.000,E1 355.584} C_DIS
LIN {X 0.128,Y -442.898,Z 902.774,A 0.000,B 0.000,C 90.000,E1 355.241} C_DIS
LIN {X 0.057,Y -447.296,Z 902.772,A 0.000,B 0.000,C 90.000,E1 354.951} C_DIS
LIN {X -0.153,Y -451.215,Z 902.771,A 0.000,B 0.000,C 90.000,E1 354.780} C_DIS
LIN {X -0.194,Y -461.571,Z 902.768,A 0.000,B 0.000,C 90.000,E1 354.318} C_DIS
LIN {X 0.130,Y -471.786,Z 902.766,A 0.000,B 0.000,C 90.000,E1 353.799} C_DIS
LIN {X -0.171,Y -484.862,Z 902.762,A 0.000,B 0.000,C 90.000,E1 353.166} C_DIS
LIN {X -0.151,Y -496.444,Z 902.758,A 0.000,B 0.000,C 90.000,E1 352.527} C_DIS
LIN {X -0.159,Y -504.580,Z 902.756,A 0.000,B 0.000,C 90.000,E1 352.064} C_DIS
LIN {X -0.092,Y -515.606,Z 902.752,A 0.000,B 0.000,C 90.000,E1 351.376} C_DIS
LIN {X -0.078,Y -521.842,Z 902.750,A 0.000,B 0.000,C 90.000,E1 350.971} C_DIS
LIN {X -0.206,Y -529.531,Z 902.747,A 0.000,B 0.000,C 90.000,E1 350.443} C_DIS
LIN {X -0.011,Y -536.801,Z 902.744,A 0.000,B 0.000,C 90.000,E1 349.859} C_DIS
LIN {X 0.224,Y -545.223,Z 902.740,A 0.000,B 0.000,C 90.000,E1 349.106} C_DIS
LIN {X -0.090,Y -550.593,Z 902.737,A 0.000,B 0.000,C 90.000,E1 348.634} C_DIS
LIN {X -0.032,Y -556.852,Z 902.733,A 0.000,B 0.000,C 90.000,E1 347.993} C_DIS
LIN {X -0.058,Y -560.622,Z 902.731,A 0.000,B 0.000,C 90.000,E1 347.589} C_DIS
LIN {X 0.264,Y -566.407,Z 902.727,A 0.000,B 0.000,C 90.000,E1 346.881} C_DIS
LIN {X -0.317,Y -573.180,Z 902.723,A 0.000,B 0.000,C 90.000,E1 346.117} C_DIS
LIN {X 0.175,Y -580.168,Z 902.717,A 0.000,B 0.000,C 90.000,E1 345.117} C_DIS
LIN {X -0.128,Y -585.778,Z 902.713,A 0.000,B 0.000,C 90.000,E1 344.338} C_DIS
LIN {X -0.298,Y -590.051,Z 902.709,A 0.000,B 0.000,C 90.000,E1 343.685} C_DIS
LIN {X -0.062,Y -596.370,Z 902.703,A 0.000,B 0.000,C 90.000,E1 342.598} C_DIS
LIN {X -0.144,Y -600.069,Z 902.700,A 0.000,B 0.000,C 90.000,E1 341.945} C_DIS
LIN {X -0.295,Y -605.019,Z 902.695,A 0.000,B 0.000,C 90.000,E1 341.040} C_DIS
LIN {X -0.151,Y -608.999,Z 902.690,A 0.000,B 0.000,C 90.000,E1 340.242} C_DIS
LIN {X 0.041,Y -612.910,Z 902.686,A 0.000,B 0.000,C 90.000,E1 339.444} C_DIS
LIN {X 0.021,Y -617.800,Z 902.680,A 0.000,B 0.000,C 90.000,E1 338.411} C_DIS
LIN {X 0.286,Y -622.387,Z 902.674,A 0.000,B 0.000,C 90.000,E1 337.358} C_DIS
LIN {X 0.047,Y -627.660,Z 902.667,A 0.000,B 0.000,C 90.000,E1 336.102} C_DIS
LIN {X -0.179,Y -629.647,Z 902.664,A 0.000,B 0.000,C 90.000,E1 335.613} C_DIS
LIN {X -0.070,Y -633.380,Z 902.659,A 0.000,B 0.000,C 90.000,E1 334.588} C_DIS
LIN {X 0.098,Y -636.993,Z 902.653,A 0.000,B 0.000,C 90.000,E1 333.563} C_DIS
LIN {X 0.022,Y -640.320,Z 902.648,A 0.000,B 0.000,C 90.000,E1 332.564} C_DIS
LIN {X 0.009,Y -643.320,Z 902.642,A 0.000,B 0.000,C 90.000,E1 331.563} C_DIS
LIN {X -0.109,Y -647.496,Z 902.634,A 0.000,B 0.000,C 90.000,E1 330.078} C_DIS
LIN {X 0.072,Y -650.779,Z 902.627,A 0.000,B 0.000,C 90.000,E1 328.820} C_DIS
LIN {X -0.345,Y -653.195,Z 902.621,A 0.000,B 0.000,C 90.000,E1 327.867} C_DIS
LIN {X 0.177,Y -655.330,Z 902.616,A 0.000,B 0.000,C 90.000,E1 326.834} C_DIS
LIN {X -0.180,Y -657.147,Z 902.610,A 0.000,B 0.000,C 90.000,E1 325.881} C_DIS
LIN {X -0.053,Y -659.135,Z 902.604,A 0.000,B 0.000,C 90.000,E1 324.642} C_DIS
LIN {X -0.049,Y -660.737,Z 902.597,A 0.000,B 0.000,C 90.000,E1 323.417} C_DIS
LIN {X 0.028,Y -661.807,Z 902.591,A 0.000,B 0.000,C 90.000,E1 322.431} C_DIS
LIN {X -0.028,Y -663.010,Z 902.585,A 0.000,B 0.000,C 90.000,E1 321.215} C_DIS
LIN {X 0.041,Y -664.168,Z 902.578,A 0.000,B 0.000,C 90.000,E1 319.989} C_DIS
LIN {X 0.024,Y -665.809,Z 902.568,A 0.000,B 0.000,C 90.000,E1 318.286} C_DIS
LIN {X 0.056,Y -666.825,Z 902.563,A 0.000,B 0.000,C 90.000,E1 317.310} C_DIS
LIN {X 0.062,Y -667.869,Z 902.557,A 0.000,B 0.000,C 90.000,E1 316.338} C_DIS
LIN {X -0.379,Y -668.764,Z 902.552,A 0.000,B 0.000,C 90.000,E1 315.405} C_DIS
LIN {X -0.335,Y -669.922,Z 902.545,A 0.000,B 0.000,C 90.000,E1 314.190} C_DIS
LIN {X -0.314,Y -670.295,Z 902.543,A 0.000,B 0.000,C 90.000,E1 313.704} C_DIS
LIN {X 0.235,Y -671.451,Z 902.536,A 0.000,B 0.000,C 90.000,E1 312.447} C_DIS
LIN {X 0.353,Y -672.600,Z 902.529,A 0.000,B 0.000,C 90.000,E1 311.229} C_DIS
LIN {X 0.070,Y -673.742,Z 902.521,A 0.000,B 0.000,C 90.000,E1 309.806} C_DIS
LIN {X -0.196,Y -674.916,Z 902.513,A 0.000,B 0.000,C 90.000,E1 308.382} C_DIS
LIN {X 0.073,Y -675.831,Z 902.507,A 0.000,B 0.000,C 90.000,E1 307.156} C_DIS
LIN {X -0.044,Y -676.599,Z 902.500,A 0.000,B 0.000,C 90.000,E1 305.964} C_DIS
LIN {X 0.245,Y -677.240,Z 902.493,A 0.000,B 0.000,C 90.000,E1 304.739} C_DIS
LIN {X -0.303,Y -678.419,Z 902.481,A 0.000,B 0.000,C 90.000,E1 302.625} C_DIS
LIN {X -0.234,Y -679.996,Z 902.469,A 0.000,B 0.000,C 90.000,E1 300.463} C_DIS
LIN {X -0.193,Y -682.901,Z 902.453,A 0.000,B 0.000,C 90.000,E1 297.590} C_DIS
LIN {X 0.215,Y -685.736,Z 902.441,A 0.000,B 0.000,C 90.000,E1 295.412} C_DIS
LIN {X 0.187,Y -686.942,Z 902.436,A 0.000,B 0.000,C 90.000,E1 294.463} C_DIS
LIN {X 0.172,Y -687.943,Z 902.431,A 0.000,B 0.000,C 90.000,E1 293.515} C_DIS
LIN {X -0.285,Y -688.099,Z 902.428,A 0.000,B 0.000,C 90.000,E1 293.078} C_DIS
LIN {X -0.064,Y -688.011,Z 902.427,A 0.000,B 0.000,C 90.000,E1 292.823} C_DIS
LIN {X 0.115,Y -687.168,Z 902.424,A 0.000,B 0.000,C 90.000,E1 292.333} C_DIS
LIN {X 0.074,Y -686.409,Z 902.423,A 0.000,B 0.000,C 90.000,E1 292.099} C_DIS
LIN {X -0.136,Y -683.244,Z 902.420,A 0.000,B 0.000,C 90.000,E1 291.642} C_DIS
LIN {X -0.286,Y -682.285,Z 902.420,A 0.000,B 0.000,C 90.000,E1 291.535} C_DIS
LIN {X -0.184,Y -681.041,Z 902.419,A 0.000,B 0.000,C 90.000,E1 291.408} C_DIS
LIN {X -0.052,Y -679.138,Z 902.418,A 0.000,B 0.000,C 90.000,E1 291.280} C_DIS
